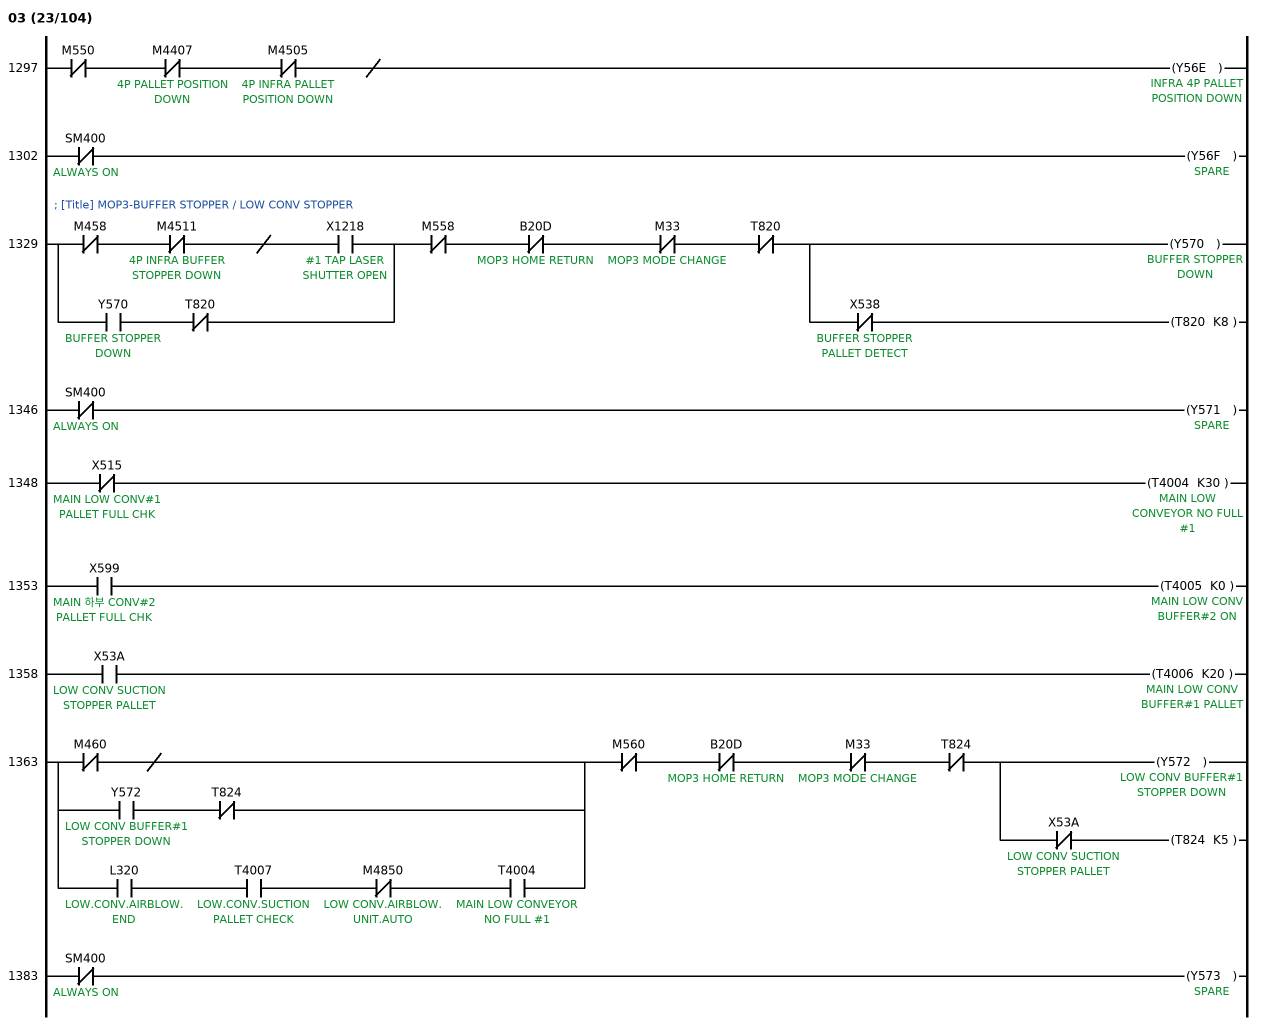
1297  LDI     M550
      ANI     M4407  ; 4P PALLET POSITION DOWN
      ANI     M4505  ; 4P INFRA PALLET POSITION DOWN
      INV
      OUT     Y56E  ; INFRA 4P PALLET POSITION DOWN
1302  LDI     SM400  ; ALWAYS ON
      OUT     Y56F  ; SPARE
; [Title] MOP3-BUFFER STOPPER / LOW CONV STOPPER
1329  LDI     M458
      ANI     M4511  ; 4P INFRA BUFFER STOPPER DOWN
      INV
      AND     X1218  ; #1 TAP LASER SHUTTER OPEN
      LD      Y570  ; BUFFER STOPPER DOWN
      ANI     T820
      ORB
      ANI     M558
      ANI     B20D  ; MOP3 HOME RETURN
      ANI     M33  ; MOP3 MODE CHANGE
      ANI     T820
      OUT     Y570  ; BUFFER STOPPER DOWN
      ANI     X538  ; BUFFER STOPPER PALLET DETECT
      OUT     T820 K8
1346  LDI     SM400  ; ALWAYS ON
      OUT     Y571  ; SPARE
1348  LDI     X515  ; MAIN LOW CONV#1 PALLET FULL CHK
      OUT     T4004 K30  ; MAIN LOW CONVEYOR NO FULL #1
1353  LD      X599  ; MAIN 하부 CONV#2 PALLET FULL CHK
      OUT     T4005 K0  ; MAIN LOW CONV BUFFER#2 ON
1358  LD      X53A  ; LOW CONV SUCTION STOPPER PALLET
      OUT     T4006 K20  ; MAIN LOW CONV BUFFER#1 PALLET
1363  LDI     M460
      INV
      LD      Y572  ; LOW CONV BUFFER#1 STOPPER DOWN
      ANI     T824
      ORB
      LD      L320  ; LOW.CONV.AIRBLOW.END
      AND     T4007  ; LOW.CONV.SUCTION PALLET CHECK
      ANI     M4850  ; LOW CONV.AIRBLOW.UNIT.AUTO
      AND     T4004  ; MAIN LOW CONVEYOR NO FULL #1
      ORB
      ANI     M560
      ANI     B20D  ; MOP3 HOME RETURN
      ANI     M33  ; MOP3 MODE CHANGE
      ANI     T824
      OUT     Y572  ; LOW CONV BUFFER#1 STOPPER DOWN
      ANI     X53A  ; LOW CONV SUCTION STOPPER PALLET
      OUT     T824 K5
1383  LDI     SM400  ; ALWAYS ON
      OUT     Y573  ; SPARE
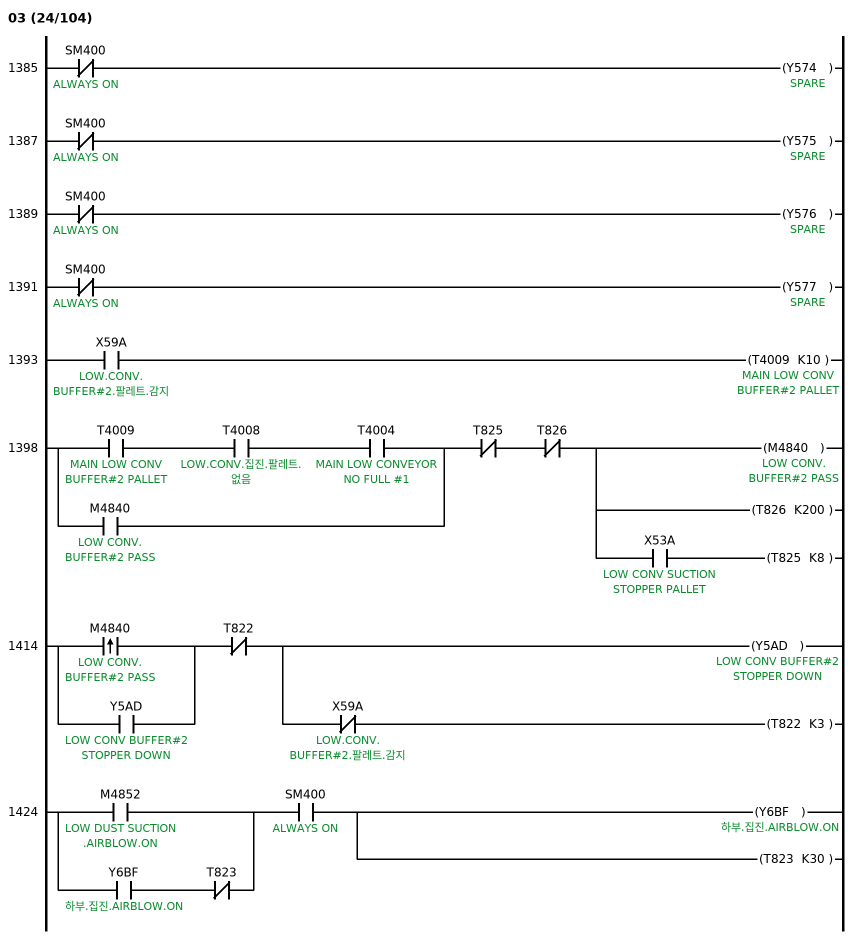
1385  LDI     SM400  ; ALWAYS ON
      OUT     Y574  ; SPARE
1387  LDI     SM400  ; ALWAYS ON
      OUT     Y575  ; SPARE
1389  LDI     SM400  ; ALWAYS ON
      OUT     Y576  ; SPARE
1391  LDI     SM400  ; ALWAYS ON
      OUT     Y577  ; SPARE
1393  LD      X59A  ; LOW.CONV.BUFFER#2.팔레트.감지
      OUT     T4009 K10  ; MAIN LOW CONV BUFFER#2 PALLET
1398  LD      T4009  ; MAIN LOW CONV BUFFER#2 PALLET
      AND     T4008  ; LOW.CONV.집진.팔레트.없음
      AND     T4004  ; MAIN LOW CONVEYOR NO FULL #1
      OR      M4840  ; LOW CONV. BUFFER#2 PASS
      ANI     T825
      ANI     T826
      OUT     M4840  ; LOW CONV. BUFFER#2 PASS
      OUT     T826 K200
      AND     X53A  ; LOW CONV SUCTION STOPPER PALLET
      OUT     T825 K8
1414  LDP     M4840  ; LOW CONV. BUFFER#2 PASS
      OR      Y5AD  ; LOW CONV BUFFER#2 STOPPER DOWN
      ANI     T822
      OUT     Y5AD  ; LOW CONV BUFFER#2 STOPPER DOWN
      ANI     X59A  ; LOW.CONV.BUFFER#2.팔레트.감지
      OUT     T822 K3
1424  LD      M4852  ; LOW DUST SUCTION .AIRBLOW.ON
      LD      Y6BF  ; 하부.집진.AIRBLOW.ON
      ANI     T823
      ORB
      AND     SM400  ; ALWAYS ON
      OUT     Y6BF  ; 하부.집진.AIRBLOW.ON
      OUT     T823 K30
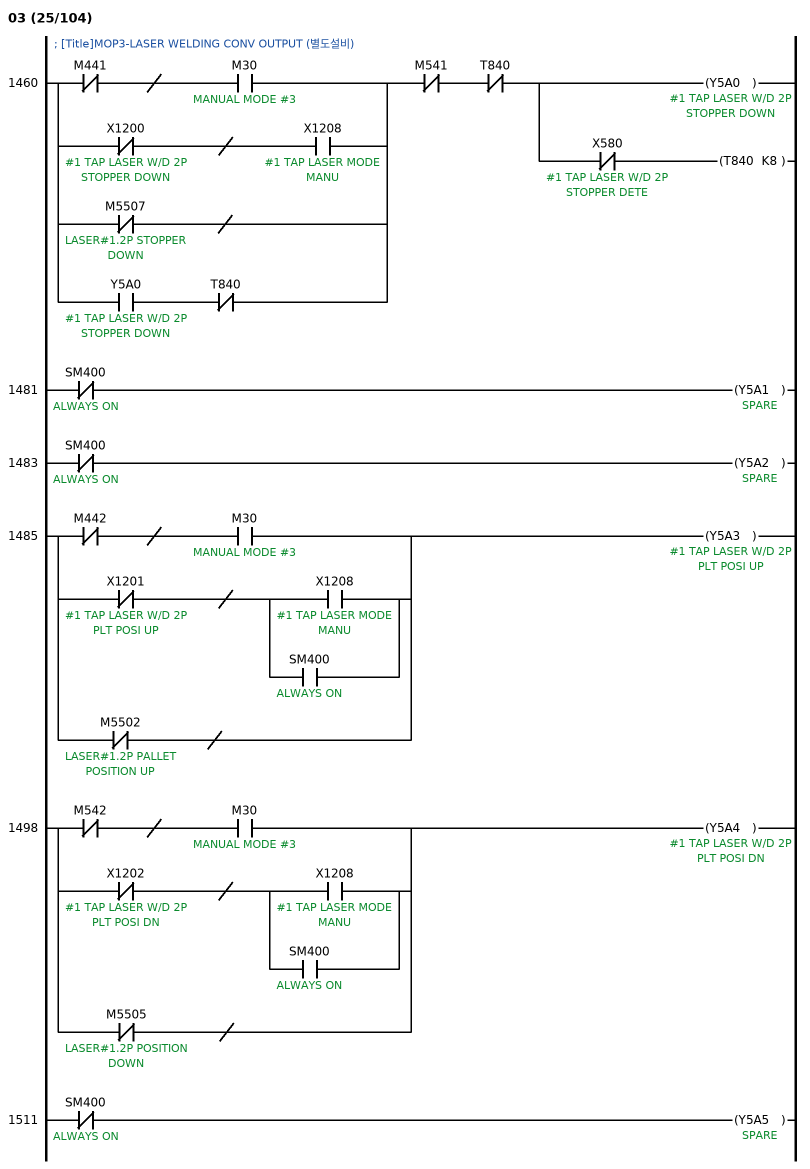
; [Title]MOP3-LASER WELDING CONV OUTPUT (별도설비)
1460  LDI     M441
      INV
      AND     M30  ; MANUAL MODE #3
      LDI     X1200  ; #1 TAP LASER W/D 2P STOPPER DOWN
      INV
      AND     X1208  ; #1 TAP LASER MODE MANU
      ORB
      LDI     M5507  ; LASER#1.2P STOPPER DOWN
      INV
      ORB
      LD      Y5A0  ; #1 TAP LASER W/D 2P STOPPER DOWN
      ANI     T840
      ORB
      ANI     M541
      ANI     T840
      OUT     Y5A0  ; #1 TAP LASER W/D 2P STOPPER DOWN
      ANI     X580  ; #1 TAP LASER W/D 2P STOPPER DETE
      OUT     T840 K8
1481  LDI     SM400  ; ALWAYS ON
      OUT     Y5A1  ; SPARE
1483  LDI     SM400  ; ALWAYS ON
      OUT     Y5A2  ; SPARE
1485  LDI     M442
      INV
      AND     M30  ; MANUAL MODE #3
      LDI     X1201  ; #1 TAP LASER W/D 2P PLT POSI UP
      INV
      LD      X1208  ; #1 TAP LASER MODE MANU
      OR      SM400  ; ALWAYS ON
      ANB
      ORB
      LDI     M5502  ; LASER#1.2P PALLET POSITION UP
      INV
      ORB
      OUT     Y5A3  ; #1 TAP LASER W/D 2P PLT POSI UP
1498  LDI     M542
      INV
      AND     M30  ; MANUAL MODE #3
      LDI     X1202  ; #1 TAP LASER W/D 2P PLT POSI DN
      INV
      LD      X1208  ; #1 TAP LASER MODE MANU
      OR      SM400  ; ALWAYS ON
      ANB
      ORB
      LDI     M5505  ; LASER#1.2P POSITION DOWN
      INV
      ORB
      OUT     Y5A4  ; #1 TAP LASER W/D 2P PLT POSI DN
1511  LDI     SM400  ; ALWAYS ON
      OUT     Y5A5  ; SPARE
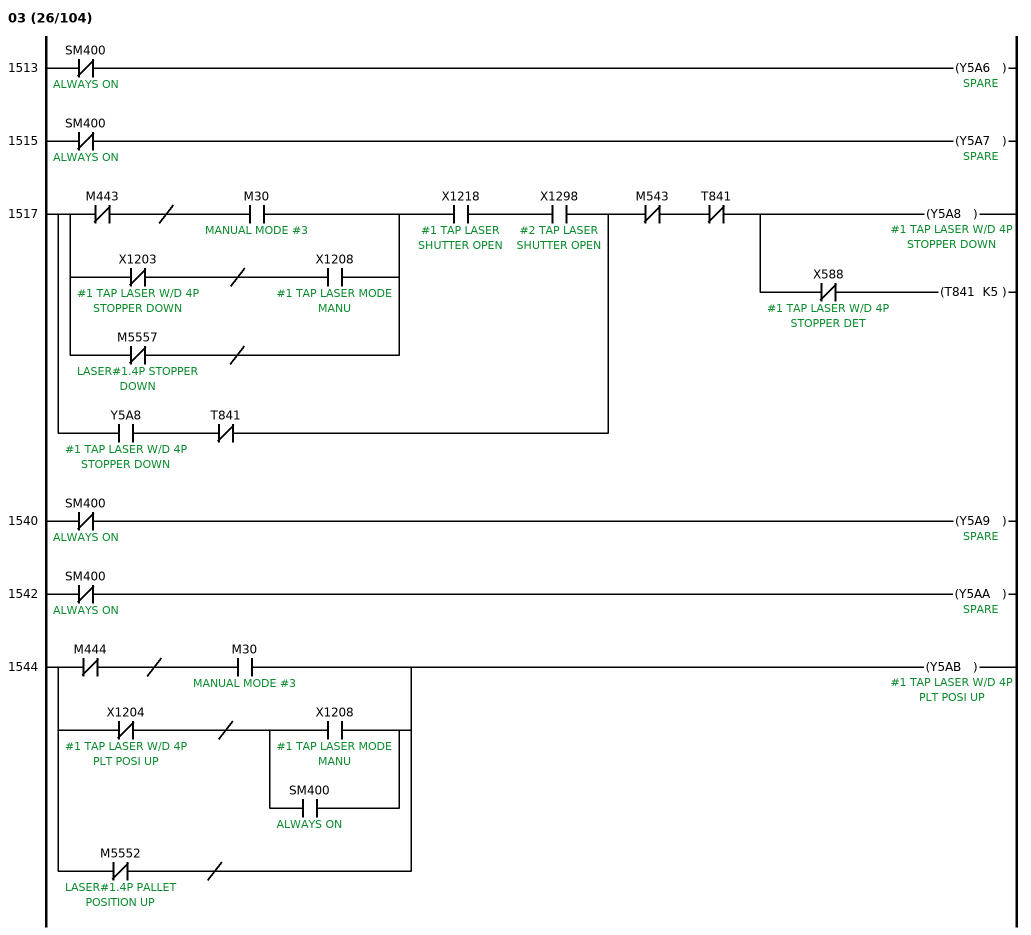
1513  LDI     SM400  ; ALWAYS ON
      OUT     Y5A6  ; SPARE
1515  LDI     SM400  ; ALWAYS ON
      OUT     Y5A7  ; SPARE
1517  LDI     M443
      INV
      AND     M30  ; MANUAL MODE #3
      LDI     X1203  ; #1 TAP LASER W/D 4P STOPPER DOWN
      INV
      AND     X1208  ; #1 TAP LASER MODE MANU
      ORB
      LDI     M5557  ; LASER#1.4P STOPPER DOWN
      INV
      ORB
      AND     X1218  ; #1 TAP LASER SHUTTER OPEN
      AND     X1298  ; #2 TAP LASER SHUTTER OPEN
      LD      Y5A8  ; #1 TAP LASER W/D 4P STOPPER DOWN
      ANI     T841
      ORB
      ANI     M543
      ANI     T841
      OUT     Y5A8  ; #1 TAP LASER W/D 4P STOPPER DOWN
      ANI     X588  ; #1 TAP LASER W/D 4P STOPPER DET
      OUT     T841 K5
1540  LDI     SM400  ; ALWAYS ON
      OUT     Y5A9  ; SPARE
1542  LDI     SM400  ; ALWAYS ON
      OUT     Y5AA  ; SPARE
1544  LDI     M444
      INV
      AND     M30  ; MANUAL MODE #3
      LDI     X1204  ; #1 TAP LASER W/D 4P PLT POSI UP
      INV
      LD      X1208  ; #1 TAP LASER MODE MANU
      OR      SM400  ; ALWAYS ON
      ANB
      ORB
      LDI     M5552  ; LASER#1.4P PALLET POSITION UP
      INV
      ORB
      OUT     Y5AB  ; #1 TAP LASER W/D 4P PLT POSI UP
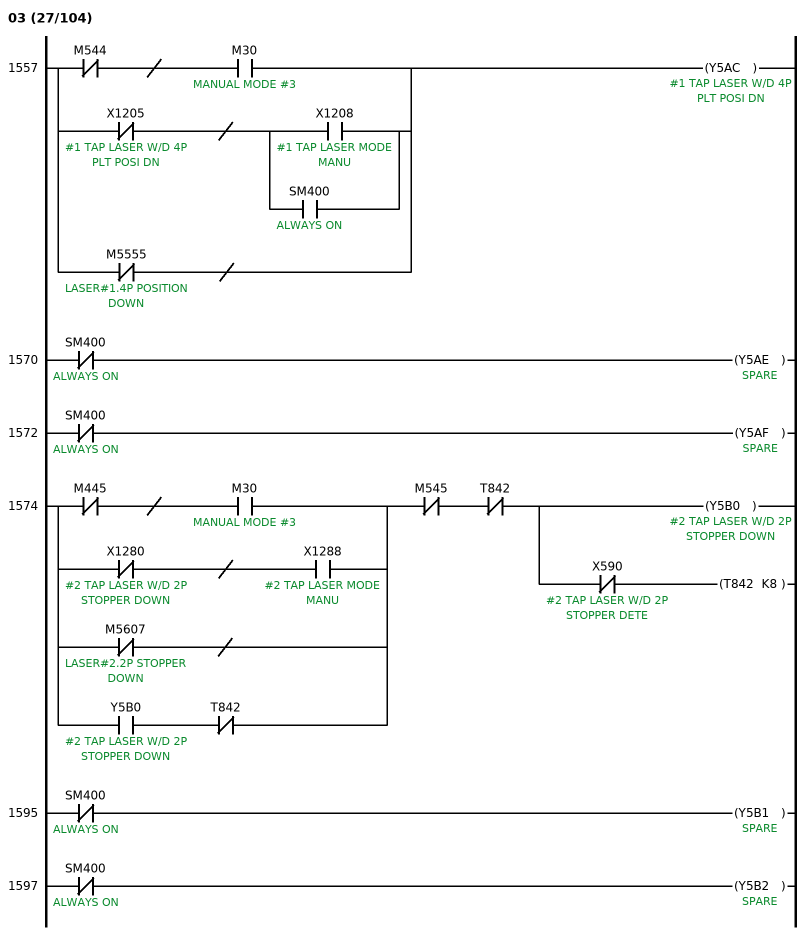
1557  LDI     M544
      INV
      AND     M30  ; MANUAL MODE #3
      LDI     X1205  ; #1 TAP LASER W/D 4P PLT POSI DN
      INV
      LD      X1208  ; #1 TAP LASER MODE MANU
      OR      SM400  ; ALWAYS ON
      ANB
      ORB
      LDI     M5555  ; LASER#1.4P POSITION DOWN
      INV
      ORB
      OUT     Y5AC  ; #1 TAP LASER W/D 4P PLT POSI DN
1570  LDI     SM400  ; ALWAYS ON
      OUT     Y5AE  ; SPARE
1572  LDI     SM400  ; ALWAYS ON
      OUT     Y5AF  ; SPARE
1574  LDI     M445
      INV
      AND     M30  ; MANUAL MODE #3
      LDI     X1280  ; #2 TAP LASER W/D 2P STOPPER DOWN
      INV
      AND     X1288  ; #2 TAP LASER MODE MANU
      ORB
      LDI     M5607  ; LASER#2.2P STOPPER DOWN
      INV
      ORB
      LD      Y5B0  ; #2 TAP LASER W/D 2P STOPPER DOWN
      ANI     T842
      ORB
      ANI     M545
      ANI     T842
      OUT     Y5B0  ; #2 TAP LASER W/D 2P STOPPER DOWN
      ANI     X590  ; #2 TAP LASER W/D 2P STOPPER DETE
      OUT     T842 K8
1595  LDI     SM400  ; ALWAYS ON
      OUT     Y5B1  ; SPARE
1597  LDI     SM400  ; ALWAYS ON
      OUT     Y5B2  ; SPARE
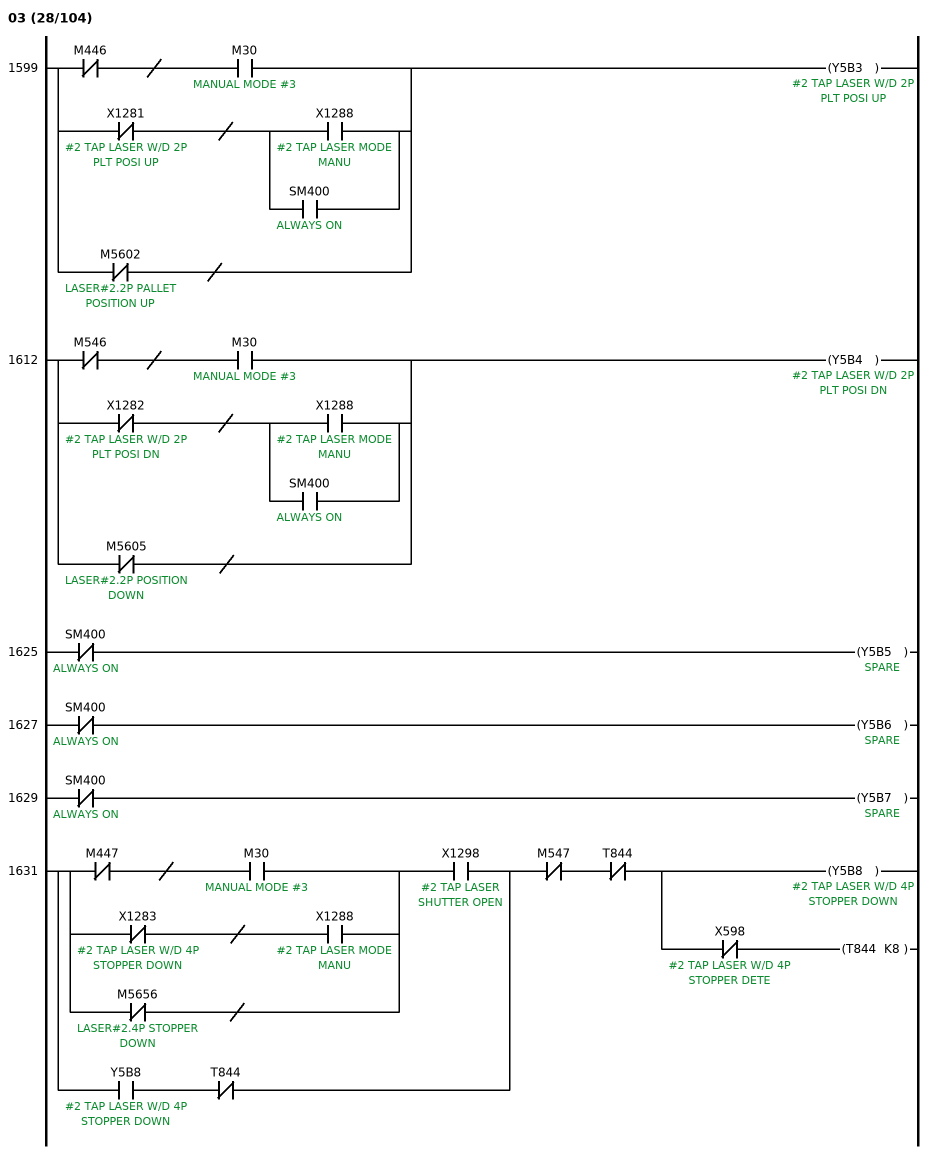
1599  LDI     M446
      INV
      AND     M30  ; MANUAL MODE #3
      LDI     X1281  ; #2 TAP LASER W/D 2P PLT POSI UP
      INV
      LD      X1288  ; #2 TAP LASER MODE MANU
      OR      SM400  ; ALWAYS ON
      ANB
      ORB
      LDI     M5602  ; LASER#2.2P PALLET POSITION UP
      INV
      ORB
      OUT     Y5B3  ; #2 TAP LASER W/D 2P PLT POSI UP
1612  LDI     M546
      INV
      AND     M30  ; MANUAL MODE #3
      LDI     X1282  ; #2 TAP LASER W/D 2P PLT POSI DN
      INV
      LD      X1288  ; #2 TAP LASER MODE MANU
      OR      SM400  ; ALWAYS ON
      ANB
      ORB
      LDI     M5605  ; LASER#2.2P POSITION DOWN
      INV
      ORB
      OUT     Y5B4  ; #2 TAP LASER W/D 2P PLT POSI DN
1625  LDI     SM400  ; ALWAYS ON
      OUT     Y5B5  ; SPARE
1627  LDI     SM400  ; ALWAYS ON
      OUT     Y5B6  ; SPARE
1629  LDI     SM400  ; ALWAYS ON
      OUT     Y5B7  ; SPARE
1631  LDI     M447
      INV
      AND     M30  ; MANUAL MODE #3
      LDI     X1283  ; #2 TAP LASER W/D 4P STOPPER DOWN
      INV
      AND     X1288  ; #2 TAP LASER MODE MANU
      ORB
      LDI     M5656  ; LASER#2.4P STOPPER DOWN
      INV
      ORB
      AND     X1298  ; #2 TAP LASER SHUTTER OPEN
      LD      Y5B8  ; #2 TAP LASER W/D 4P STOPPER DOWN
      ANI     T844
      ORB
      ANI     M547
      ANI     T844
      OUT     Y5B8  ; #2 TAP LASER W/D 4P STOPPER DOWN
      ANI     X598  ; #2 TAP LASER W/D 4P STOPPER DETE
      OUT     T844 K8
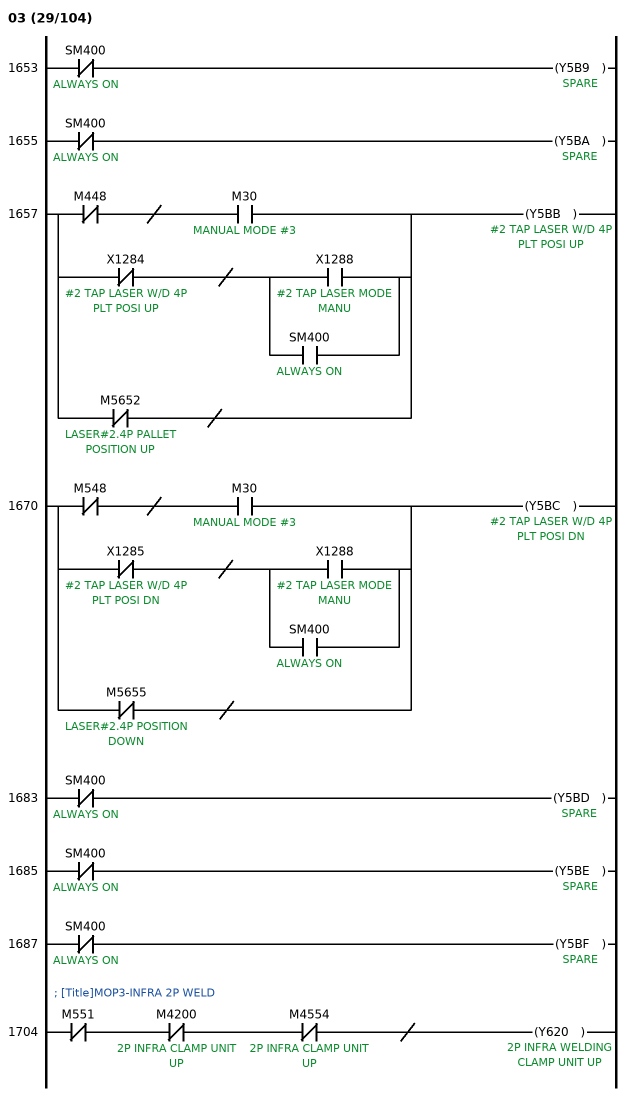
1653  LDI     SM400  ; ALWAYS ON
      OUT     Y5B9  ; SPARE
1655  LDI     SM400  ; ALWAYS ON
      OUT     Y5BA  ; SPARE
1657  LDI     M448
      INV
      AND     M30  ; MANUAL MODE #3
      LDI     X1284  ; #2 TAP LASER W/D 4P PLT POSI UP
      INV
      LD      X1288  ; #2 TAP LASER MODE MANU
      OR      SM400  ; ALWAYS ON
      ANB
      ORB
      LDI     M5652  ; LASER#2.4P PALLET POSITION UP
      INV
      ORB
      OUT     Y5BB  ; #2 TAP LASER W/D 4P PLT POSI UP
1670  LDI     M548
      INV
      AND     M30  ; MANUAL MODE #3
      LDI     X1285  ; #2 TAP LASER W/D 4P PLT POSI DN
      INV
      LD      X1288  ; #2 TAP LASER MODE MANU
      OR      SM400  ; ALWAYS ON
      ANB
      ORB
      LDI     M5655  ; LASER#2.4P POSITION DOWN
      INV
      ORB
      OUT     Y5BC  ; #2 TAP LASER W/D 4P PLT POSI DN
1683  LDI     SM400  ; ALWAYS ON
      OUT     Y5BD  ; SPARE
1685  LDI     SM400  ; ALWAYS ON
      OUT     Y5BE  ; SPARE
1687  LDI     SM400  ; ALWAYS ON
      OUT     Y5BF  ; SPARE
; [Title]MOP3-INFRA 2P WELD
1704  LDI     M551
      ANI     M4200  ; 2P INFRA CLAMP UNIT UP
      ANI     M4554  ; 2P INFRA CLAMP UNIT UP
      INV
      OUT     Y620  ; 2P INFRA WELDING CLAMP UNIT UP
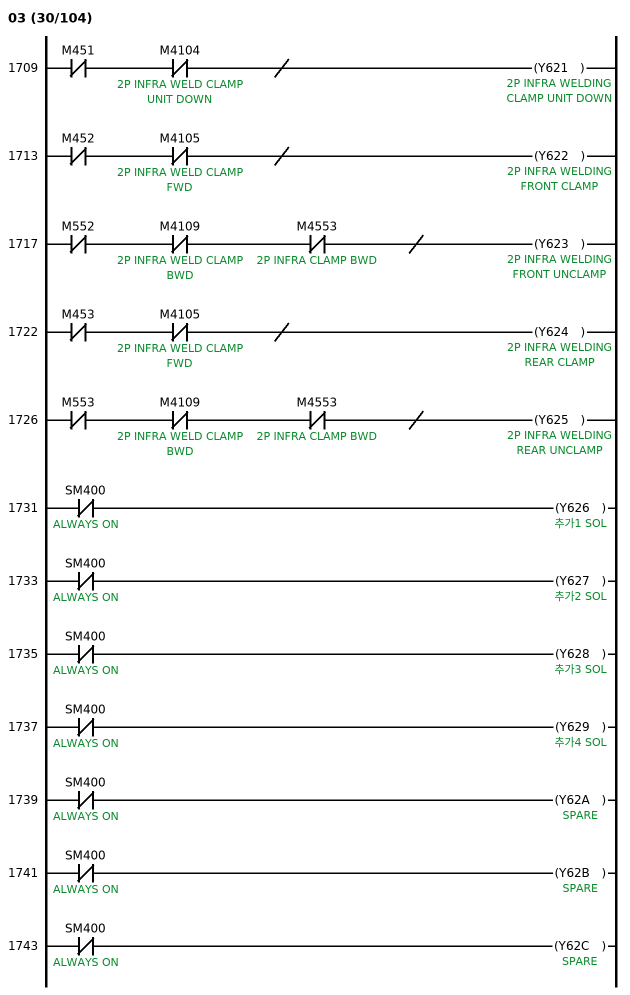
1709  LDI     M451
      ANI     M4104  ; 2P INFRA WELD CLAMP UNIT DOWN
      INV
      OUT     Y621  ; 2P INFRA WELDING CLAMP UNIT DOWN
1713  LDI     M452
      ANI     M4105  ; 2P INFRA WELD CLAMP FWD
      INV
      OUT     Y622  ; 2P INFRA WELDING FRONT CLAMP
1717  LDI     M552
      ANI     M4109  ; 2P INFRA WELD CLAMP BWD
      ANI     M4553  ; 2P INFRA CLAMP BWD
      INV
      OUT     Y623  ; 2P INFRA WELDING FRONT UNCLAMP
1722  LDI     M453
      ANI     M4105  ; 2P INFRA WELD CLAMP FWD
      INV
      OUT     Y624  ; 2P INFRA WELDING REAR CLAMP
1726  LDI     M553
      ANI     M4109  ; 2P INFRA WELD CLAMP BWD
      ANI     M4553  ; 2P INFRA CLAMP BWD
      INV
      OUT     Y625  ; 2P INFRA WELDING REAR UNCLAMP
1731  LDI     SM400  ; ALWAYS ON
      OUT     Y626  ; 추가1 SOL
1733  LDI     SM400  ; ALWAYS ON
      OUT     Y627  ; 추가2 SOL
1735  LDI     SM400  ; ALWAYS ON
      OUT     Y628  ; 추가3 SOL
1737  LDI     SM400  ; ALWAYS ON
      OUT     Y629  ; 추가4 SOL
1739  LDI     SM400  ; ALWAYS ON
      OUT     Y62A  ; SPARE
1741  LDI     SM400  ; ALWAYS ON
      OUT     Y62B  ; SPARE
1743  LDI     SM400  ; ALWAYS ON
      OUT     Y62C  ; SPARE
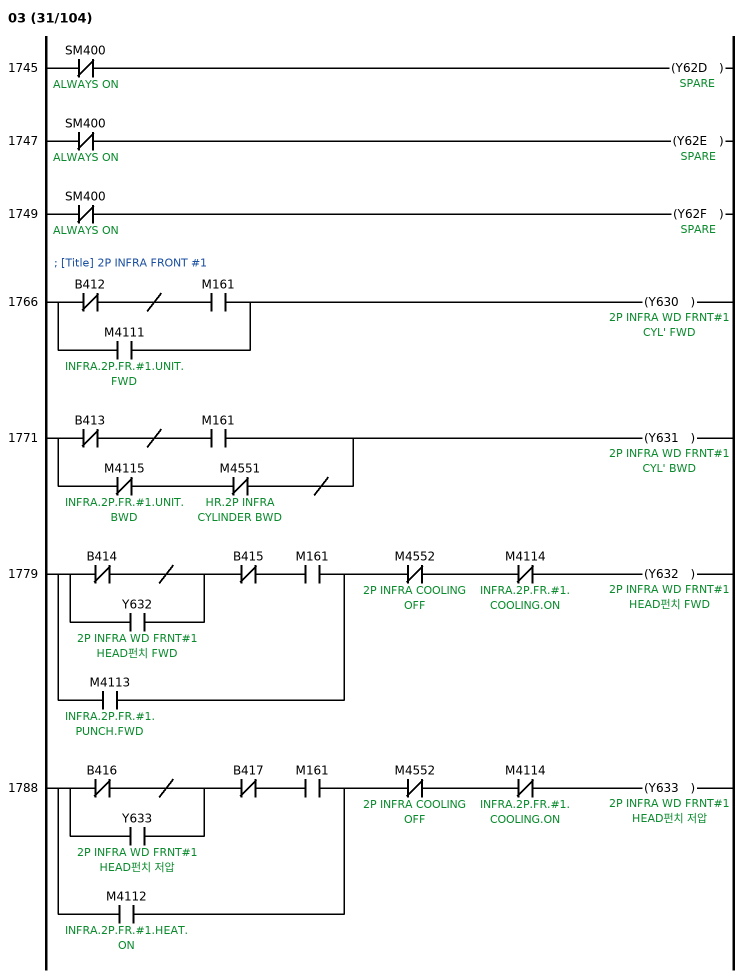
1745  LDI     SM400  ; ALWAYS ON
      OUT     Y62D  ; SPARE
1747  LDI     SM400  ; ALWAYS ON
      OUT     Y62E  ; SPARE
1749  LDI     SM400  ; ALWAYS ON
      OUT     Y62F  ; SPARE
; [Title] 2P INFRA FRONT #1
1766  LDI     B412
      INV
      AND     M161
      OR      M4111  ; INFRA.2P.FR.#1.UNIT.FWD
      OUT     Y630  ; 2P INFRA WD FRNT#1 CYL' FWD
1771  LDI     B413
      INV
      AND     M161
      LDI     M4115  ; INFRA.2P.FR.#1.UNIT.BWD
      ANI     M4551  ; HR.2P INFRA CYLINDER BWD
      INV
      ORB
      OUT     Y631  ; 2P INFRA WD FRNT#1 CYL' BWD
1779  LDI     B414
      INV
      OR      Y632  ; 2P INFRA WD FRNT#1 HEAD펀치 FWD
      ANI     B415
      AND     M161
      OR      M4113  ; INFRA.2P.FR.#1.PUNCH.FWD
      ANI     M4552  ; 2P INFRA COOLING OFF
      ANI     M4114  ; INFRA.2P.FR.#1.COOLING.ON
      OUT     Y632  ; 2P INFRA WD FRNT#1 HEAD펀치 FWD
1788  LDI     B416
      INV
      OR      Y633  ; 2P INFRA WD FRNT#1 HEAD펀치 저압
      ANI     B417
      AND     M161
      OR      M4112  ; INFRA.2P.FR.#1.HEAT.ON
      ANI     M4552  ; 2P INFRA COOLING OFF
      ANI     M4114  ; INFRA.2P.FR.#1.COOLING.ON
      OUT     Y633  ; 2P INFRA WD FRNT#1 HEAD펀치 저압
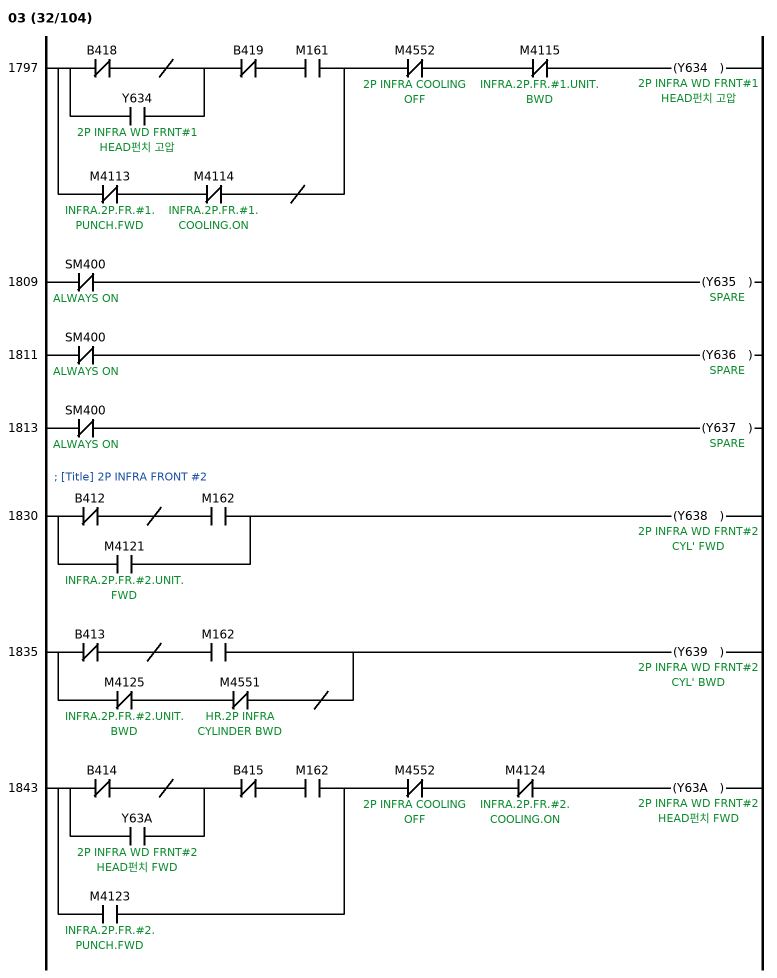
1797  LDI     B418
      INV
      OR      Y634  ; 2P INFRA WD FRNT#1 HEAD펀치 고압
      ANI     B419
      AND     M161
      LDI     M4113  ; INFRA.2P.FR.#1.PUNCH.FWD
      ANI     M4114  ; INFRA.2P.FR.#1.COOLING.ON
      INV
      ORB
      ANI     M4552  ; 2P INFRA COOLING OFF
      ANI     M4115  ; INFRA.2P.FR.#1.UNIT.BWD
      OUT     Y634  ; 2P INFRA WD FRNT#1 HEAD펀치 고압
1809  LDI     SM400  ; ALWAYS ON
      OUT     Y635  ; SPARE
1811  LDI     SM400  ; ALWAYS ON
      OUT     Y636  ; SPARE
1813  LDI     SM400  ; ALWAYS ON
      OUT     Y637  ; SPARE
; [Title] 2P INFRA FRONT #2
1830  LDI     B412
      INV
      AND     M162
      OR      M4121  ; INFRA.2P.FR.#2.UNIT.FWD
      OUT     Y638  ; 2P INFRA WD FRNT#2 CYL' FWD
1835  LDI     B413
      INV
      AND     M162
      LDI     M4125  ; INFRA.2P.FR.#2.UNIT.BWD
      ANI     M4551  ; HR.2P INFRA CYLINDER BWD
      INV
      ORB
      OUT     Y639  ; 2P INFRA WD FRNT#2 CYL' BWD
1843  LDI     B414
      INV
      OR      Y63A  ; 2P INFRA WD FRNT#2 HEAD펀치 FWD
      ANI     B415
      AND     M162
      OR      M4123  ; INFRA.2P.FR.#2.PUNCH.FWD
      ANI     M4552  ; 2P INFRA COOLING OFF
      ANI     M4124  ; INFRA.2P.FR.#2.COOLING.ON
      OUT     Y63A  ; 2P INFRA WD FRNT#2 HEAD펀치 FWD
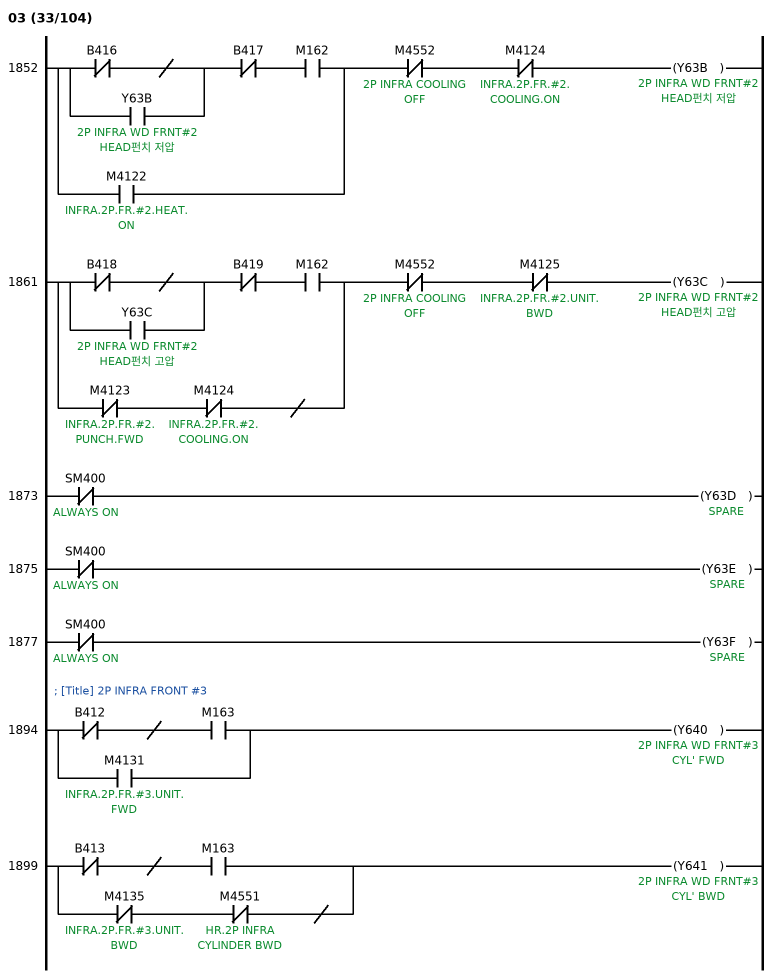
1852  LDI     B416
      INV
      OR      Y63B  ; 2P INFRA WD FRNT#2 HEAD펀치 저압
      ANI     B417
      AND     M162
      OR      M4122  ; INFRA.2P.FR.#2.HEAT.ON
      ANI     M4552  ; 2P INFRA COOLING OFF
      ANI     M4124  ; INFRA.2P.FR.#2.COOLING.ON
      OUT     Y63B  ; 2P INFRA WD FRNT#2 HEAD펀치 저압
1861  LDI     B418
      INV
      OR      Y63C  ; 2P INFRA WD FRNT#2 HEAD펀치 고압
      ANI     B419
      AND     M162
      LDI     M4123  ; INFRA.2P.FR.#2.PUNCH.FWD
      ANI     M4124  ; INFRA.2P.FR.#2.COOLING.ON
      INV
      ORB
      ANI     M4552  ; 2P INFRA COOLING OFF
      ANI     M4125  ; INFRA.2P.FR.#2.UNIT.BWD
      OUT     Y63C  ; 2P INFRA WD FRNT#2 HEAD펀치 고압
1873  LDI     SM400  ; ALWAYS ON
      OUT     Y63D  ; SPARE
1875  LDI     SM400  ; ALWAYS ON
      OUT     Y63E  ; SPARE
1877  LDI     SM400  ; ALWAYS ON
      OUT     Y63F  ; SPARE
; [Title] 2P INFRA FRONT #3
1894  LDI     B412
      INV
      AND     M163
      OR      M4131  ; INFRA.2P.FR.#3.UNIT.FWD
      OUT     Y640  ; 2P INFRA WD FRNT#3 CYL' FWD
1899  LDI     B413
      INV
      AND     M163
      LDI     M4135  ; INFRA.2P.FR.#3.UNIT.BWD
      ANI     M4551  ; HR.2P INFRA CYLINDER BWD
      INV
      ORB
      OUT     Y641  ; 2P INFRA WD FRNT#3 CYL' BWD
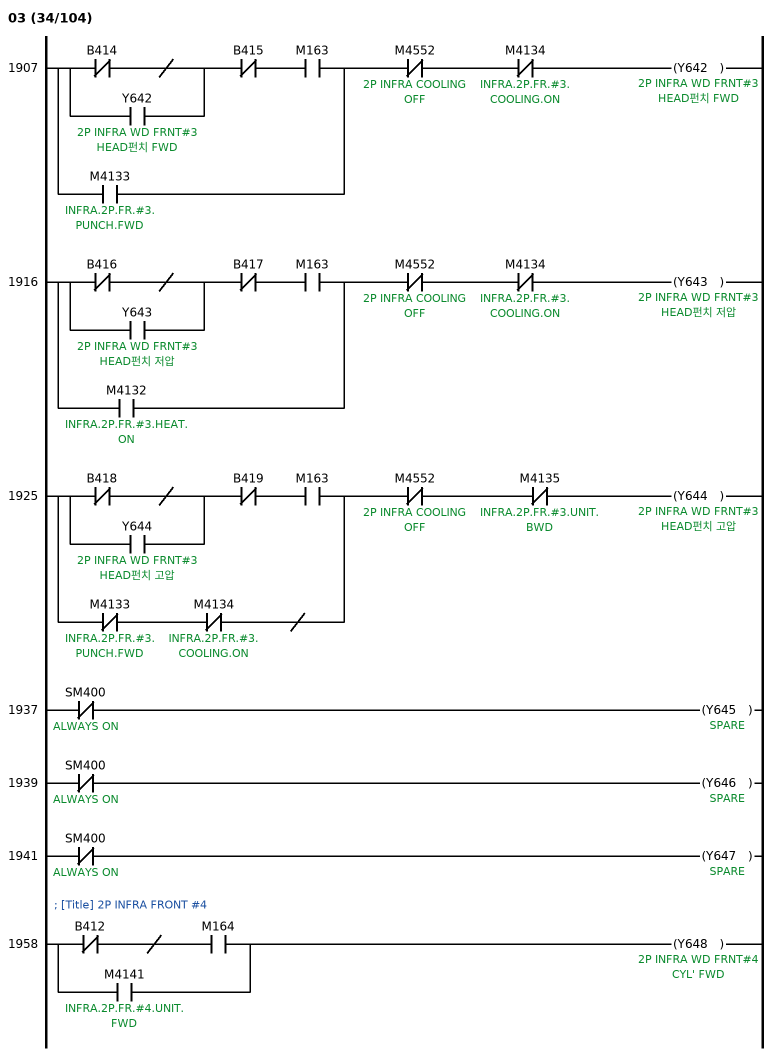
1907  LDI     B414
      INV
      OR      Y642  ; 2P INFRA WD FRNT#3 HEAD펀치 FWD
      ANI     B415
      AND     M163
      OR      M4133  ; INFRA.2P.FR.#3.PUNCH.FWD
      ANI     M4552  ; 2P INFRA COOLING OFF
      ANI     M4134  ; INFRA.2P.FR.#3.COOLING.ON
      OUT     Y642  ; 2P INFRA WD FRNT#3 HEAD펀치 FWD
1916  LDI     B416
      INV
      OR      Y643  ; 2P INFRA WD FRNT#3 HEAD펀치 저압
      ANI     B417
      AND     M163
      OR      M4132  ; INFRA.2P.FR.#3.HEAT.ON
      ANI     M4552  ; 2P INFRA COOLING OFF
      ANI     M4134  ; INFRA.2P.FR.#3.COOLING.ON
      OUT     Y643  ; 2P INFRA WD FRNT#3 HEAD펀치 저압
1925  LDI     B418
      INV
      OR      Y644  ; 2P INFRA WD FRNT#3 HEAD펀치 고압
      ANI     B419
      AND     M163
      LDI     M4133  ; INFRA.2P.FR.#3.PUNCH.FWD
      ANI     M4134  ; INFRA.2P.FR.#3.COOLING.ON
      INV
      ORB
      ANI     M4552  ; 2P INFRA COOLING OFF
      ANI     M4135  ; INFRA.2P.FR.#3.UNIT.BWD
      OUT     Y644  ; 2P INFRA WD FRNT#3 HEAD펀치 고압
1937  LDI     SM400  ; ALWAYS ON
      OUT     Y645  ; SPARE
1939  LDI     SM400  ; ALWAYS ON
      OUT     Y646  ; SPARE
1941  LDI     SM400  ; ALWAYS ON
      OUT     Y647  ; SPARE
; [Title] 2P INFRA FRONT #4
1958  LDI     B412
      INV
      AND     M164
      OR      M4141  ; INFRA.2P.FR.#4.UNIT.FWD
      OUT     Y648  ; 2P INFRA WD FRNT#4 CYL' FWD
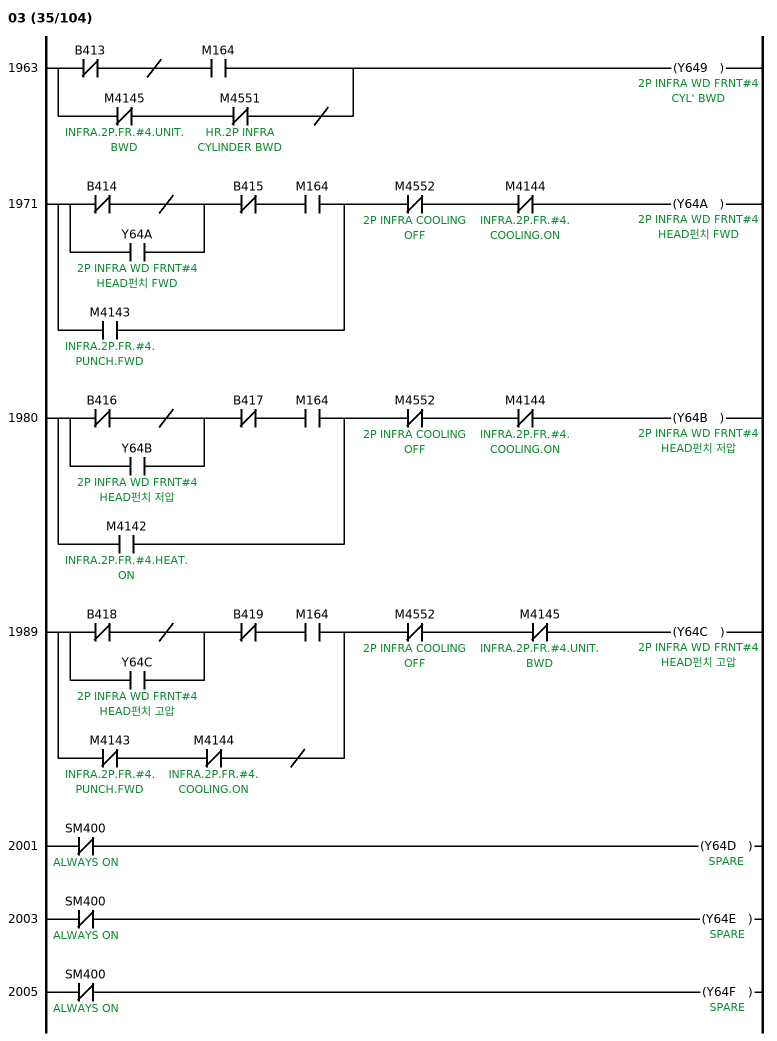
1963  LDI     B413
      INV
      AND     M164
      LDI     M4145  ; INFRA.2P.FR.#4.UNIT.BWD
      ANI     M4551  ; HR.2P INFRA CYLINDER BWD
      INV
      ORB
      OUT     Y649  ; 2P INFRA WD FRNT#4 CYL' BWD
1971  LDI     B414
      INV
      OR      Y64A  ; 2P INFRA WD FRNT#4 HEAD펀치 FWD
      ANI     B415
      AND     M164
      OR      M4143  ; INFRA.2P.FR.#4.PUNCH.FWD
      ANI     M4552  ; 2P INFRA COOLING OFF
      ANI     M4144  ; INFRA.2P.FR.#4.COOLING.ON
      OUT     Y64A  ; 2P INFRA WD FRNT#4 HEAD펀치 FWD
1980  LDI     B416
      INV
      OR      Y64B  ; 2P INFRA WD FRNT#4 HEAD펀치 저압
      ANI     B417
      AND     M164
      OR      M4142  ; INFRA.2P.FR.#4.HEAT.ON
      ANI     M4552  ; 2P INFRA COOLING OFF
      ANI     M4144  ; INFRA.2P.FR.#4.COOLING.ON
      OUT     Y64B  ; 2P INFRA WD FRNT#4 HEAD펀치 저압
1989  LDI     B418
      INV
      OR      Y64C  ; 2P INFRA WD FRNT#4 HEAD펀치 고압
      ANI     B419
      AND     M164
      LDI     M4143  ; INFRA.2P.FR.#4.PUNCH.FWD
      ANI     M4144  ; INFRA.2P.FR.#4.COOLING.ON
      INV
      ORB
      ANI     M4552  ; 2P INFRA COOLING OFF
      ANI     M4145  ; INFRA.2P.FR.#4.UNIT.BWD
      OUT     Y64C  ; 2P INFRA WD FRNT#4 HEAD펀치 고압
2001  LDI     SM400  ; ALWAYS ON
      OUT     Y64D  ; SPARE
2003  LDI     SM400  ; ALWAYS ON
      OUT     Y64E  ; SPARE
2005  LDI     SM400  ; ALWAYS ON
      OUT     Y64F  ; SPARE
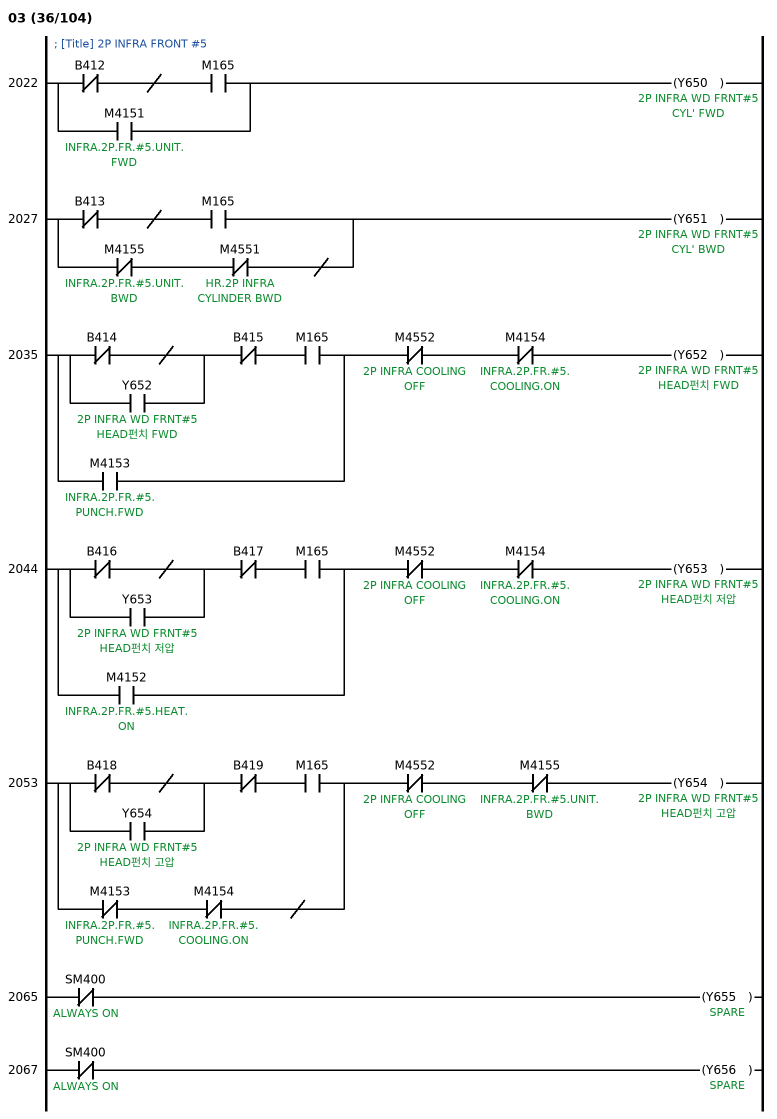
; [Title] 2P INFRA FRONT #5
2022  LDI     B412
      INV
      AND     M165
      OR      M4151  ; INFRA.2P.FR.#5.UNIT.FWD
      OUT     Y650  ; 2P INFRA WD FRNT#5 CYL' FWD
2027  LDI     B413
      INV
      AND     M165
      LDI     M4155  ; INFRA.2P.FR.#5.UNIT.BWD
      ANI     M4551  ; HR.2P INFRA CYLINDER BWD
      INV
      ORB
      OUT     Y651  ; 2P INFRA WD FRNT#5 CYL' BWD
2035  LDI     B414
      INV
      OR      Y652  ; 2P INFRA WD FRNT#5 HEAD펀치 FWD
      ANI     B415
      AND     M165
      OR      M4153  ; INFRA.2P.FR.#5.PUNCH.FWD
      ANI     M4552  ; 2P INFRA COOLING OFF
      ANI     M4154  ; INFRA.2P.FR.#5.COOLING.ON
      OUT     Y652  ; 2P INFRA WD FRNT#5 HEAD펀치 FWD
2044  LDI     B416
      INV
      OR      Y653  ; 2P INFRA WD FRNT#5 HEAD펀치 저압
      ANI     B417
      AND     M165
      OR      M4152  ; INFRA.2P.FR.#5.HEAT.ON
      ANI     M4552  ; 2P INFRA COOLING OFF
      ANI     M4154  ; INFRA.2P.FR.#5.COOLING.ON
      OUT     Y653  ; 2P INFRA WD FRNT#5 HEAD펀치 저압
2053  LDI     B418
      INV
      OR      Y654  ; 2P INFRA WD FRNT#5 HEAD펀치 고압
      ANI     B419
      AND     M165
      LDI     M4153  ; INFRA.2P.FR.#5.PUNCH.FWD
      ANI     M4154  ; INFRA.2P.FR.#5.COOLING.ON
      INV
      ORB
      ANI     M4552  ; 2P INFRA COOLING OFF
      ANI     M4155  ; INFRA.2P.FR.#5.UNIT.BWD
      OUT     Y654  ; 2P INFRA WD FRNT#5 HEAD펀치 고압
2065  LDI     SM400  ; ALWAYS ON
      OUT     Y655  ; SPARE
2067  LDI     SM400  ; ALWAYS ON
      OUT     Y656  ; SPARE
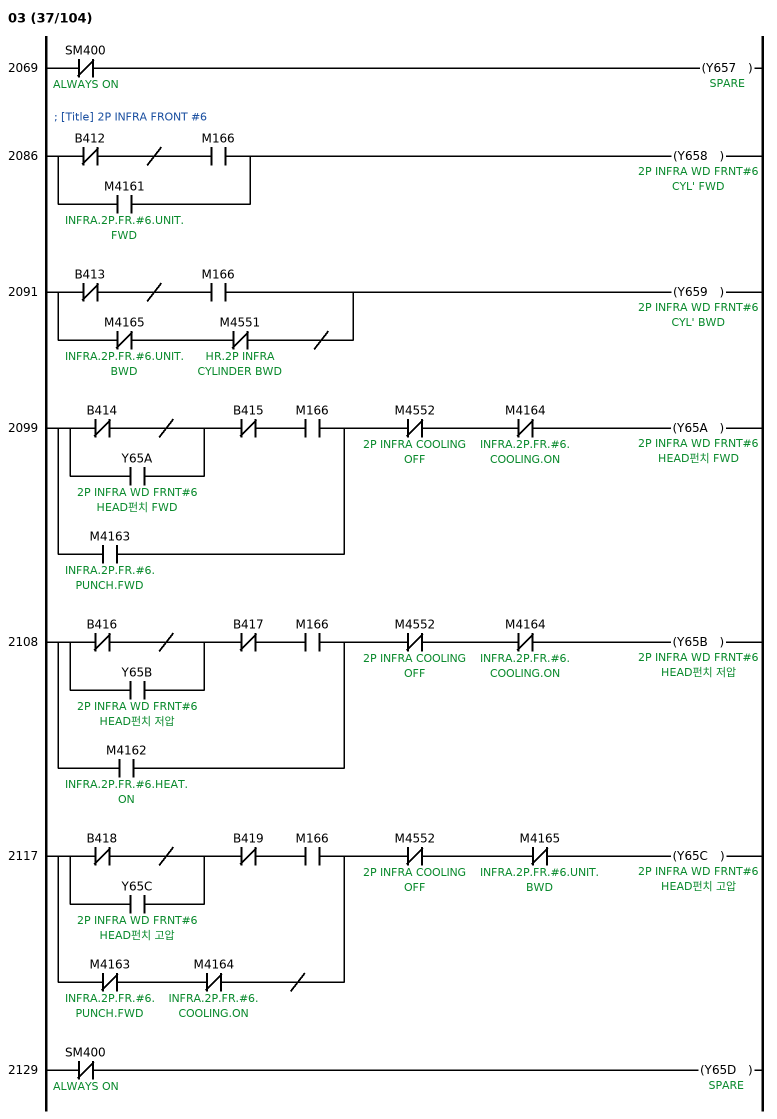
2069  LDI     SM400  ; ALWAYS ON
      OUT     Y657  ; SPARE
; [Title] 2P INFRA FRONT #6
2086  LDI     B412
      INV
      AND     M166
      OR      M4161  ; INFRA.2P.FR.#6.UNIT.FWD
      OUT     Y658  ; 2P INFRA WD FRNT#6 CYL' FWD
2091  LDI     B413
      INV
      AND     M166
      LDI     M4165  ; INFRA.2P.FR.#6.UNIT.BWD
      ANI     M4551  ; HR.2P INFRA CYLINDER BWD
      INV
      ORB
      OUT     Y659  ; 2P INFRA WD FRNT#6 CYL' BWD
2099  LDI     B414
      INV
      OR      Y65A  ; 2P INFRA WD FRNT#6 HEAD펀치 FWD
      ANI     B415
      AND     M166
      OR      M4163  ; INFRA.2P.FR.#6.PUNCH.FWD
      ANI     M4552  ; 2P INFRA COOLING OFF
      ANI     M4164  ; INFRA.2P.FR.#6.COOLING.ON
      OUT     Y65A  ; 2P INFRA WD FRNT#6 HEAD펀치 FWD
2108  LDI     B416
      INV
      OR      Y65B  ; 2P INFRA WD FRNT#6 HEAD펀치 저압
      ANI     B417
      AND     M166
      OR      M4162  ; INFRA.2P.FR.#6.HEAT.ON
      ANI     M4552  ; 2P INFRA COOLING OFF
      ANI     M4164  ; INFRA.2P.FR.#6.COOLING.ON
      OUT     Y65B  ; 2P INFRA WD FRNT#6 HEAD펀치 저압
2117  LDI     B418
      INV
      OR      Y65C  ; 2P INFRA WD FRNT#6 HEAD펀치 고압
      ANI     B419
      AND     M166
      LDI     M4163  ; INFRA.2P.FR.#6.PUNCH.FWD
      ANI     M4164  ; INFRA.2P.FR.#6.COOLING.ON
      INV
      ORB
      ANI     M4552  ; 2P INFRA COOLING OFF
      ANI     M4165  ; INFRA.2P.FR.#6.UNIT.BWD
      OUT     Y65C  ; 2P INFRA WD FRNT#6 HEAD펀치 고압
2129  LDI     SM400  ; ALWAYS ON
      OUT     Y65D  ; SPARE
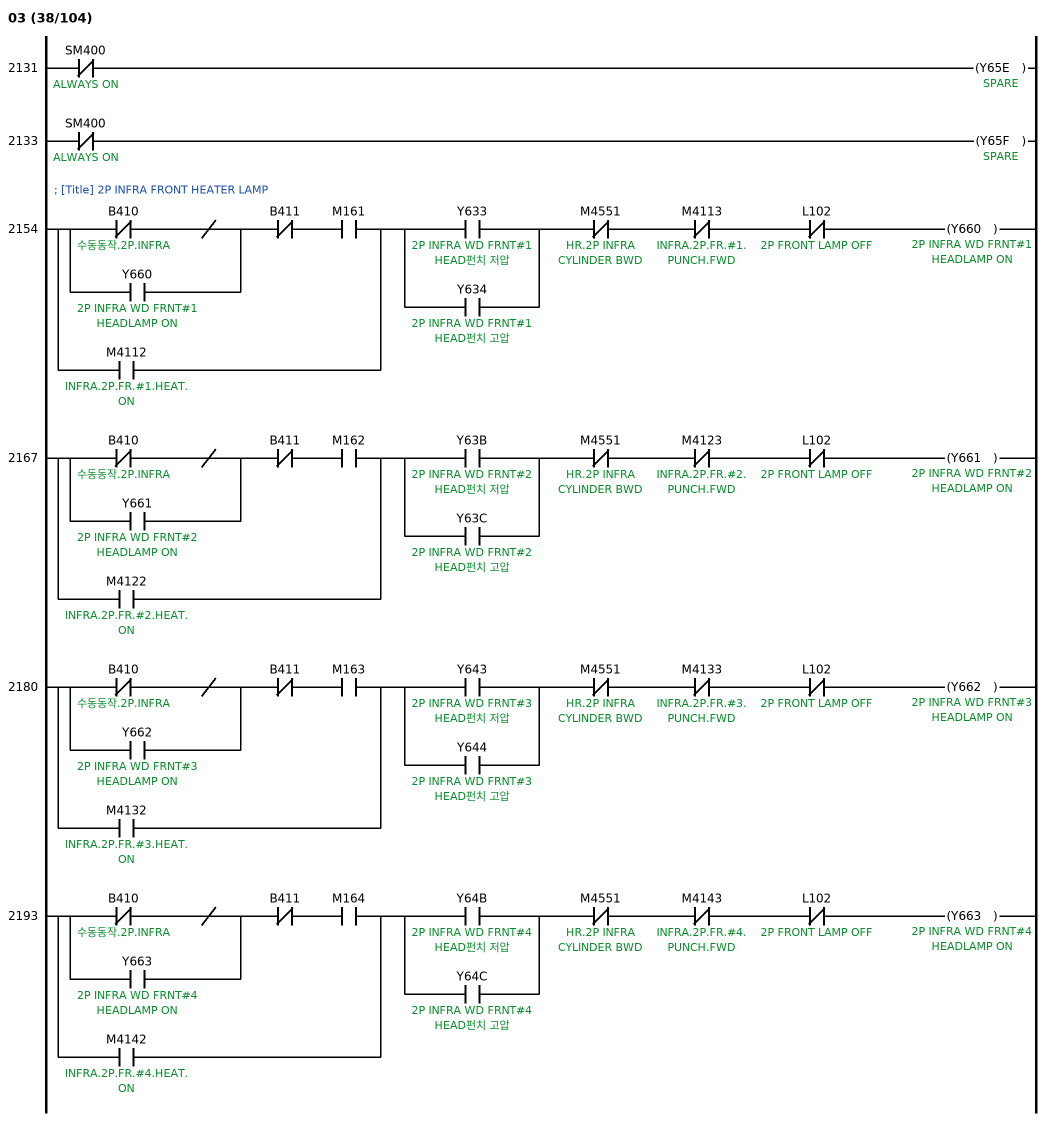
2131  LDI     SM400  ; ALWAYS ON
      OUT     Y65E  ; SPARE
2133  LDI     SM400  ; ALWAYS ON
      OUT     Y65F  ; SPARE
; [Title] 2P INFRA FRONT HEATER LAMP
2154  LDI     B410  ; 수동동작.2P.INFRA
      INV
      OR      Y660  ; 2P INFRA WD FRNT#1 HEADLAMP ON
      ANI     B411
      AND     M161
      OR      M4112  ; INFRA.2P.FR.#1.HEAT.ON
      LD      Y633  ; 2P INFRA WD FRNT#1 HEAD펀치 저압
      OR      Y634  ; 2P INFRA WD FRNT#1 HEAD펀치 고압
      ANB
      ANI     M4551  ; HR.2P INFRA CYLINDER BWD
      ANI     M4113  ; INFRA.2P.FR.#1.PUNCH.FWD
      ANI     L102  ; 2P FRONT LAMP OFF
      OUT     Y660  ; 2P INFRA WD FRNT#1 HEADLAMP ON
2167  LDI     B410  ; 수동동작.2P.INFRA
      INV
      OR      Y661  ; 2P INFRA WD FRNT#2 HEADLAMP ON
      ANI     B411
      AND     M162
      OR      M4122  ; INFRA.2P.FR.#2.HEAT.ON
      LD      Y63B  ; 2P INFRA WD FRNT#2 HEAD펀치 저압
      OR      Y63C  ; 2P INFRA WD FRNT#2 HEAD펀치 고압
      ANB
      ANI     M4551  ; HR.2P INFRA CYLINDER BWD
      ANI     M4123  ; INFRA.2P.FR.#2.PUNCH.FWD
      ANI     L102  ; 2P FRONT LAMP OFF
      OUT     Y661  ; 2P INFRA WD FRNT#2 HEADLAMP ON
2180  LDI     B410  ; 수동동작.2P.INFRA
      INV
      OR      Y662  ; 2P INFRA WD FRNT#3 HEADLAMP ON
      ANI     B411
      AND     M163
      OR      M4132  ; INFRA.2P.FR.#3.HEAT.ON
      LD      Y643  ; 2P INFRA WD FRNT#3 HEAD펀치 저압
      OR      Y644  ; 2P INFRA WD FRNT#3 HEAD펀치 고압
      ANB
      ANI     M4551  ; HR.2P INFRA CYLINDER BWD
      ANI     M4133  ; INFRA.2P.FR.#3.PUNCH.FWD
      ANI     L102  ; 2P FRONT LAMP OFF
      OUT     Y662  ; 2P INFRA WD FRNT#3 HEADLAMP ON
2193  LDI     B410  ; 수동동작.2P.INFRA
      INV
      OR      Y663  ; 2P INFRA WD FRNT#4 HEADLAMP ON
      ANI     B411
      AND     M164
      OR      M4142  ; INFRA.2P.FR.#4.HEAT.ON
      LD      Y64B  ; 2P INFRA WD FRNT#4 HEAD펀치 저압
      OR      Y64C  ; 2P INFRA WD FRNT#4 HEAD펀치 고압
      ANB
      ANI     M4551  ; HR.2P INFRA CYLINDER BWD
      ANI     M4143  ; INFRA.2P.FR.#4.PUNCH.FWD
      ANI     L102  ; 2P FRONT LAMP OFF
      OUT     Y663  ; 2P INFRA WD FRNT#4 HEADLAMP ON
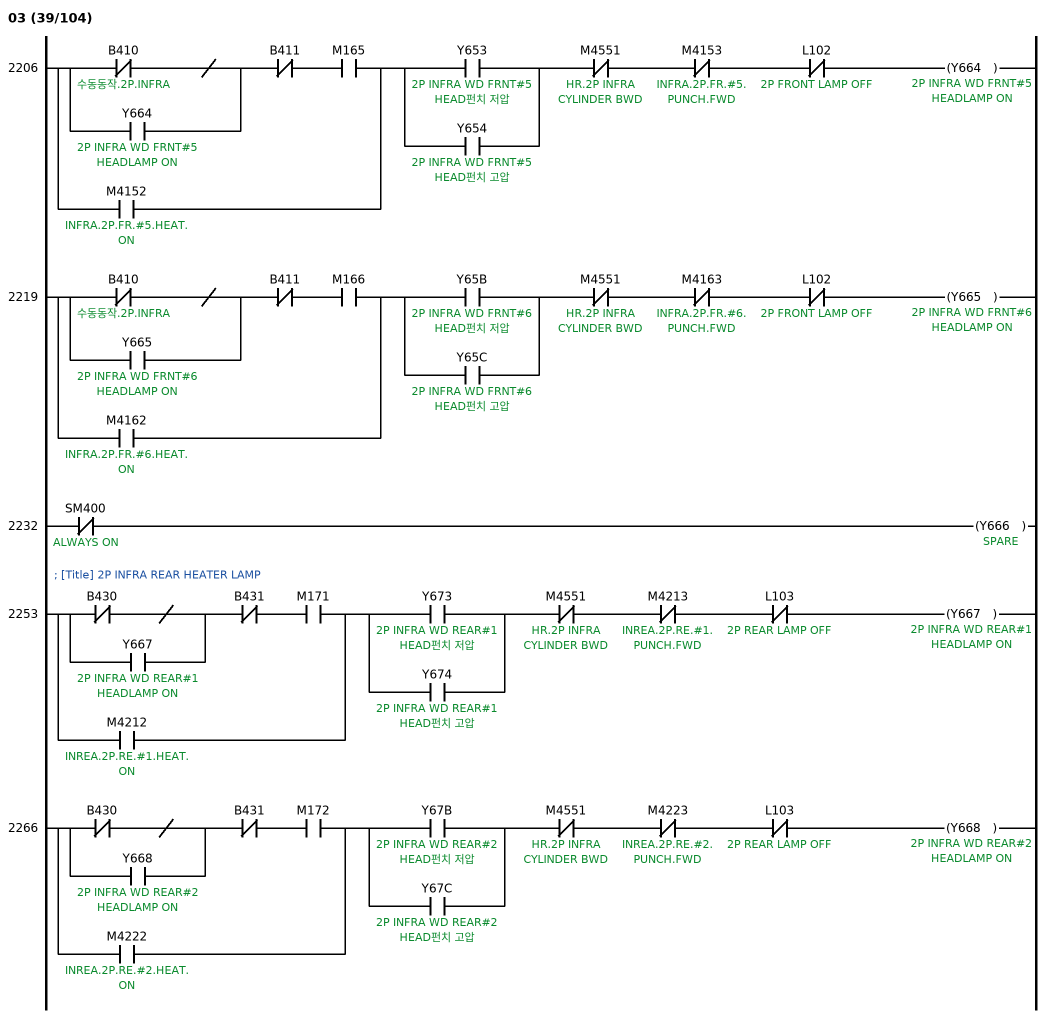
2206  LDI     B410  ; 수동동작.2P.INFRA
      INV
      OR      Y664  ; 2P INFRA WD FRNT#5 HEADLAMP ON
      ANI     B411
      AND     M165
      OR      M4152  ; INFRA.2P.FR.#5.HEAT.ON
      LD      Y653  ; 2P INFRA WD FRNT#5 HEAD펀치 저압
      OR      Y654  ; 2P INFRA WD FRNT#5 HEAD펀치 고압
      ANB
      ANI     M4551  ; HR.2P INFRA CYLINDER BWD
      ANI     M4153  ; INFRA.2P.FR.#5.PUNCH.FWD
      ANI     L102  ; 2P FRONT LAMP OFF
      OUT     Y664  ; 2P INFRA WD FRNT#5 HEADLAMP ON
2219  LDI     B410  ; 수동동작.2P.INFRA
      INV
      OR      Y665  ; 2P INFRA WD FRNT#6 HEADLAMP ON
      ANI     B411
      AND     M166
      OR      M4162  ; INFRA.2P.FR.#6.HEAT.ON
      LD      Y65B  ; 2P INFRA WD FRNT#6 HEAD펀치 저압
      OR      Y65C  ; 2P INFRA WD FRNT#6 HEAD펀치 고압
      ANB
      ANI     M4551  ; HR.2P INFRA CYLINDER BWD
      ANI     M4163  ; INFRA.2P.FR.#6.PUNCH.FWD
      ANI     L102  ; 2P FRONT LAMP OFF
      OUT     Y665  ; 2P INFRA WD FRNT#6 HEADLAMP ON
2232  LDI     SM400  ; ALWAYS ON
      OUT     Y666  ; SPARE
; [Title] 2P INFRA REAR HEATER LAMP
2253  LDI     B430
      INV
      OR      Y667  ; 2P INFRA WD REAR#1 HEADLAMP ON
      ANI     B431
      AND     M171
      OR      M4212  ; INREA.2P.RE.#1.HEAT.ON
      LD      Y673  ; 2P INFRA WD REAR#1 HEAD펀치 저압
      OR      Y674  ; 2P INFRA WD REAR#1 HEAD펀치 고압
      ANB
      ANI     M4551  ; HR.2P INFRA CYLINDER BWD
      ANI     M4213  ; INREA.2P.RE.#1.PUNCH.FWD
      ANI     L103  ; 2P REAR LAMP OFF
      OUT     Y667  ; 2P INFRA WD REAR#1 HEADLAMP ON
2266  LDI     B430
      INV
      OR      Y668  ; 2P INFRA WD REAR#2 HEADLAMP ON
      ANI     B431
      AND     M172
      OR      M4222  ; INREA.2P.RE.#2.HEAT.ON
      LD      Y67B  ; 2P INFRA WD REAR#2 HEAD펀치 저압
      OR      Y67C  ; 2P INFRA WD REAR#2 HEAD펀치 고압
      ANB
      ANI     M4551  ; HR.2P INFRA CYLINDER BWD
      ANI     M4223  ; INREA.2P.RE.#2.PUNCH.FWD
      ANI     L103  ; 2P REAR LAMP OFF
      OUT     Y668  ; 2P INFRA WD REAR#2 HEADLAMP ON
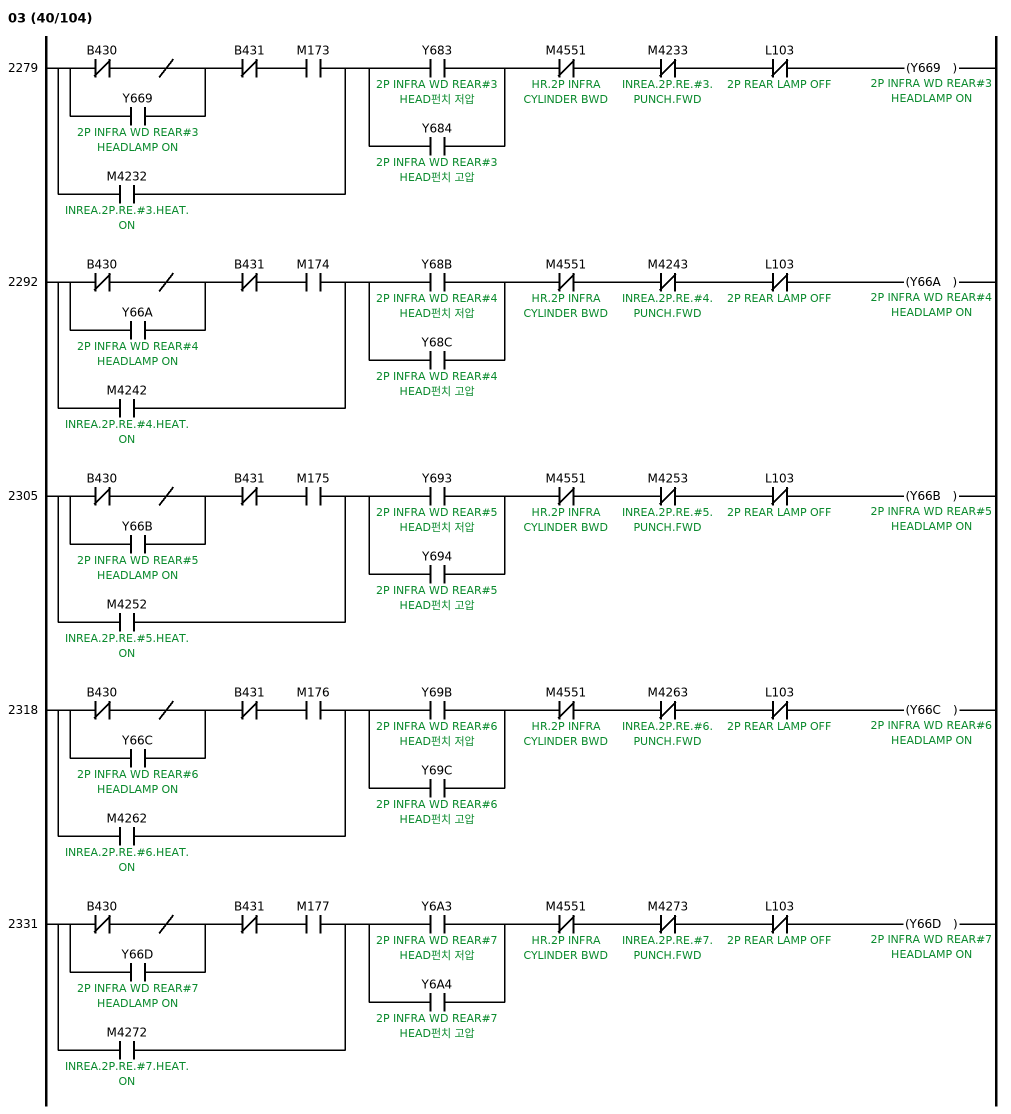
2279  LDI     B430
      INV
      OR      Y669  ; 2P INFRA WD REAR#3 HEADLAMP ON
      ANI     B431
      AND     M173
      OR      M4232  ; INREA.2P.RE.#3.HEAT.ON
      LD      Y683  ; 2P INFRA WD REAR#3 HEAD펀치 저압
      OR      Y684  ; 2P INFRA WD REAR#3 HEAD펀치 고압
      ANB
      ANI     M4551  ; HR.2P INFRA CYLINDER BWD
      ANI     M4233  ; INREA.2P.RE.#3.PUNCH.FWD
      ANI     L103  ; 2P REAR LAMP OFF
      OUT     Y669  ; 2P INFRA WD REAR#3 HEADLAMP ON
2292  LDI     B430
      INV
      OR      Y66A  ; 2P INFRA WD REAR#4 HEADLAMP ON
      ANI     B431
      AND     M174
      OR      M4242  ; INREA.2P.RE.#4.HEAT.ON
      LD      Y68B  ; 2P INFRA WD REAR#4 HEAD펀치 저압
      OR      Y68C  ; 2P INFRA WD REAR#4 HEAD펀치 고압
      ANB
      ANI     M4551  ; HR.2P INFRA CYLINDER BWD
      ANI     M4243  ; INREA.2P.RE.#4.PUNCH.FWD
      ANI     L103  ; 2P REAR LAMP OFF
      OUT     Y66A  ; 2P INFRA WD REAR#4 HEADLAMP ON
2305  LDI     B430
      INV
      OR      Y66B  ; 2P INFRA WD REAR#5 HEADLAMP ON
      ANI     B431
      AND     M175
      OR      M4252  ; INREA.2P.RE.#5.HEAT.ON
      LD      Y693  ; 2P INFRA WD REAR#5 HEAD펀치 저압
      OR      Y694  ; 2P INFRA WD REAR#5 HEAD펀치 고압
      ANB
      ANI     M4551  ; HR.2P INFRA CYLINDER BWD
      ANI     M4253  ; INREA.2P.RE.#5.PUNCH.FWD
      ANI     L103  ; 2P REAR LAMP OFF
      OUT     Y66B  ; 2P INFRA WD REAR#5 HEADLAMP ON
2318  LDI     B430
      INV
      OR      Y66C  ; 2P INFRA WD REAR#6 HEADLAMP ON
      ANI     B431
      AND     M176
      OR      M4262  ; INREA.2P.RE.#6.HEAT.ON
      LD      Y69B  ; 2P INFRA WD REAR#6 HEAD펀치 저압
      OR      Y69C  ; 2P INFRA WD REAR#6 HEAD펀치 고압
      ANB
      ANI     M4551  ; HR.2P INFRA CYLINDER BWD
      ANI     M4263  ; INREA.2P.RE.#6.PUNCH.FWD
      ANI     L103  ; 2P REAR LAMP OFF
      OUT     Y66C  ; 2P INFRA WD REAR#6 HEADLAMP ON
2331  LDI     B430
      INV
      OR      Y66D  ; 2P INFRA WD REAR#7 HEADLAMP ON
      ANI     B431
      AND     M177
      OR      M4272  ; INREA.2P.RE.#7.HEAT.ON
      LD      Y6A3  ; 2P INFRA WD REAR#7 HEAD펀치 저압
      OR      Y6A4  ; 2P INFRA WD REAR#7 HEAD펀치 고압
      ANB
      ANI     M4551  ; HR.2P INFRA CYLINDER BWD
      ANI     M4273  ; INREA.2P.RE.#7.PUNCH.FWD
      ANI     L103  ; 2P REAR LAMP OFF
      OUT     Y66D  ; 2P INFRA WD REAR#7 HEADLAMP ON
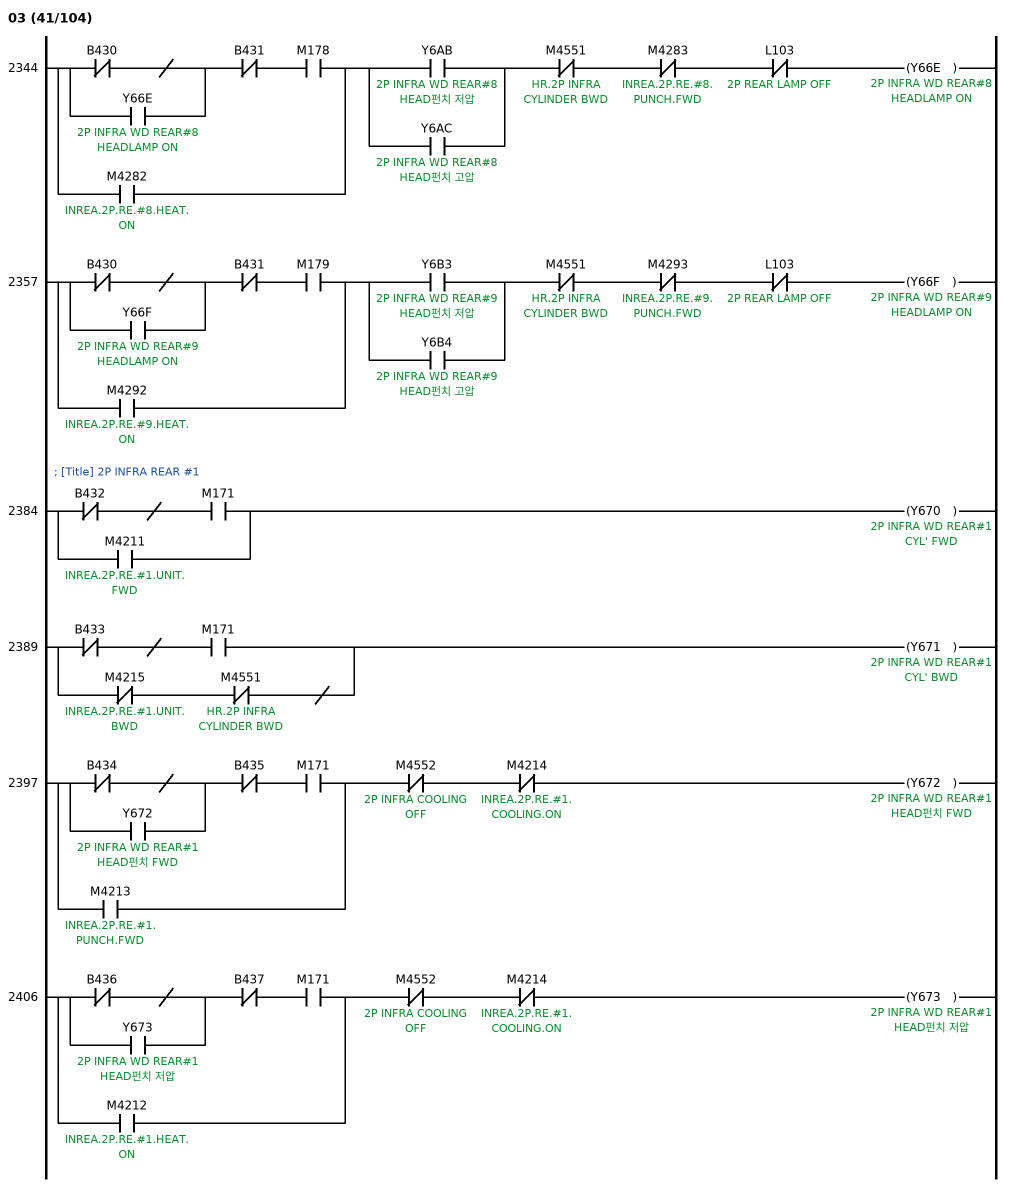
2344  LDI     B430
      INV
      OR      Y66E  ; 2P INFRA WD REAR#8 HEADLAMP ON
      ANI     B431
      AND     M178
      OR      M4282  ; INREA.2P.RE.#8.HEAT.ON
      LD      Y6AB  ; 2P INFRA WD REAR#8 HEAD펀치 저압
      OR      Y6AC  ; 2P INFRA WD REAR#8 HEAD펀치 고압
      ANB
      ANI     M4551  ; HR.2P INFRA CYLINDER BWD
      ANI     M4283  ; INREA.2P.RE.#8.PUNCH.FWD
      ANI     L103  ; 2P REAR LAMP OFF
      OUT     Y66E  ; 2P INFRA WD REAR#8 HEADLAMP ON
2357  LDI     B430
      INV
      OR      Y66F  ; 2P INFRA WD REAR#9 HEADLAMP ON
      ANI     B431
      AND     M179
      OR      M4292  ; INREA.2P.RE.#9.HEAT.ON
      LD      Y6B3  ; 2P INFRA WD REAR#9 HEAD펀치 저압
      OR      Y6B4  ; 2P INFRA WD REAR#9 HEAD펀치 고압
      ANB
      ANI     M4551  ; HR.2P INFRA CYLINDER BWD
      ANI     M4293  ; INREA.2P.RE.#9.PUNCH.FWD
      ANI     L103  ; 2P REAR LAMP OFF
      OUT     Y66F  ; 2P INFRA WD REAR#9 HEADLAMP ON
; [Title] 2P INFRA REAR #1
2384  LDI     B432
      INV
      AND     M171
      OR      M4211  ; INREA.2P.RE.#1.UNIT.FWD
      OUT     Y670  ; 2P INFRA WD REAR#1 CYL' FWD
2389  LDI     B433
      INV
      AND     M171
      LDI     M4215  ; INREA.2P.RE.#1.UNIT.BWD
      ANI     M4551  ; HR.2P INFRA CYLINDER BWD
      INV
      ORB
      OUT     Y671  ; 2P INFRA WD REAR#1 CYL' BWD
2397  LDI     B434
      INV
      OR      Y672  ; 2P INFRA WD REAR#1 HEAD펀치 FWD
      ANI     B435
      AND     M171
      OR      M4213  ; INREA.2P.RE.#1.PUNCH.FWD
      ANI     M4552  ; 2P INFRA COOLING OFF
      ANI     M4214  ; INREA.2P.RE.#1.COOLING.ON
      OUT     Y672  ; 2P INFRA WD REAR#1 HEAD펀치 FWD
2406  LDI     B436
      INV
      OR      Y673  ; 2P INFRA WD REAR#1 HEAD펀치 저압
      ANI     B437
      AND     M171
      OR      M4212  ; INREA.2P.RE.#1.HEAT.ON
      ANI     M4552  ; 2P INFRA COOLING OFF
      ANI     M4214  ; INREA.2P.RE.#1.COOLING.ON
      OUT     Y673  ; 2P INFRA WD REAR#1 HEAD펀치 저압
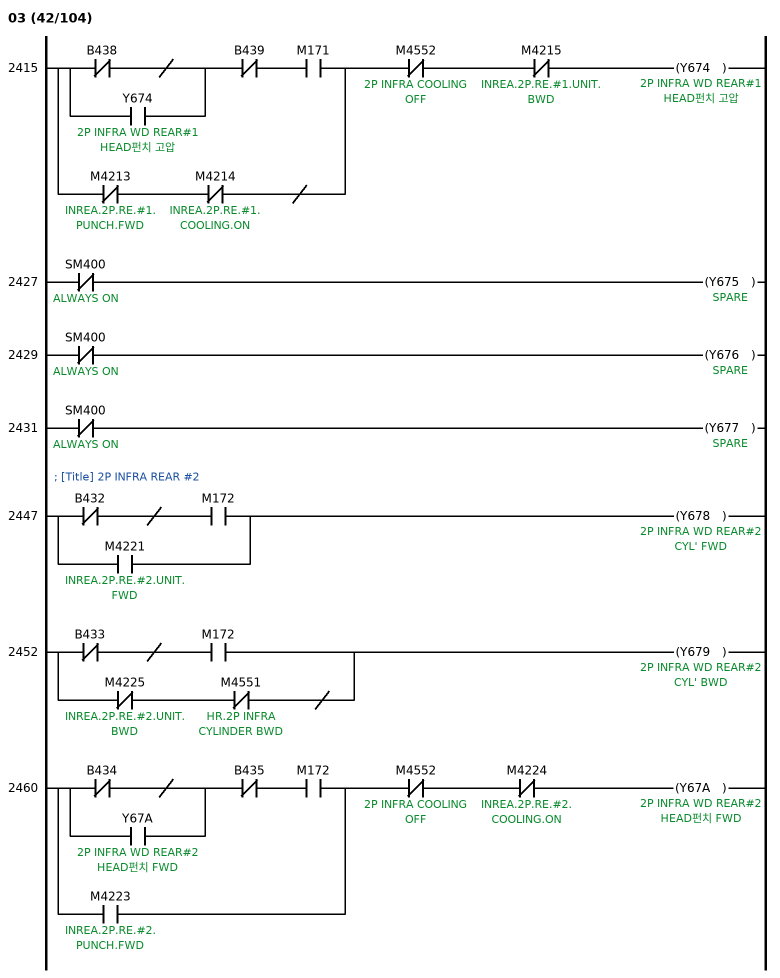
2415  LDI     B438
      INV
      OR      Y674  ; 2P INFRA WD REAR#1 HEAD펀치 고압
      ANI     B439
      AND     M171
      LDI     M4213  ; INREA.2P.RE.#1.PUNCH.FWD
      ANI     M4214  ; INREA.2P.RE.#1.COOLING.ON
      INV
      ORB
      ANI     M4552  ; 2P INFRA COOLING OFF
      ANI     M4215  ; INREA.2P.RE.#1.UNIT.BWD
      OUT     Y674  ; 2P INFRA WD REAR#1 HEAD펀치 고압
2427  LDI     SM400  ; ALWAYS ON
      OUT     Y675  ; SPARE
2429  LDI     SM400  ; ALWAYS ON
      OUT     Y676  ; SPARE
2431  LDI     SM400  ; ALWAYS ON
      OUT     Y677  ; SPARE
; [Title] 2P INFRA REAR #2
2447  LDI     B432
      INV
      AND     M172
      OR      M4221  ; INREA.2P.RE.#2.UNIT.FWD
      OUT     Y678  ; 2P INFRA WD REAR#2 CYL' FWD
2452  LDI     B433
      INV
      AND     M172
      LDI     M4225  ; INREA.2P.RE.#2.UNIT.BWD
      ANI     M4551  ; HR.2P INFRA CYLINDER BWD
      INV
      ORB
      OUT     Y679  ; 2P INFRA WD REAR#2 CYL' BWD
2460  LDI     B434
      INV
      OR      Y67A  ; 2P INFRA WD REAR#2 HEAD펀치 FWD
      ANI     B435
      AND     M172
      OR      M4223  ; INREA.2P.RE.#2.PUNCH.FWD
      ANI     M4552  ; 2P INFRA COOLING OFF
      ANI     M4224  ; INREA.2P.RE.#2.COOLING.ON
      OUT     Y67A  ; 2P INFRA WD REAR#2 HEAD펀치 FWD
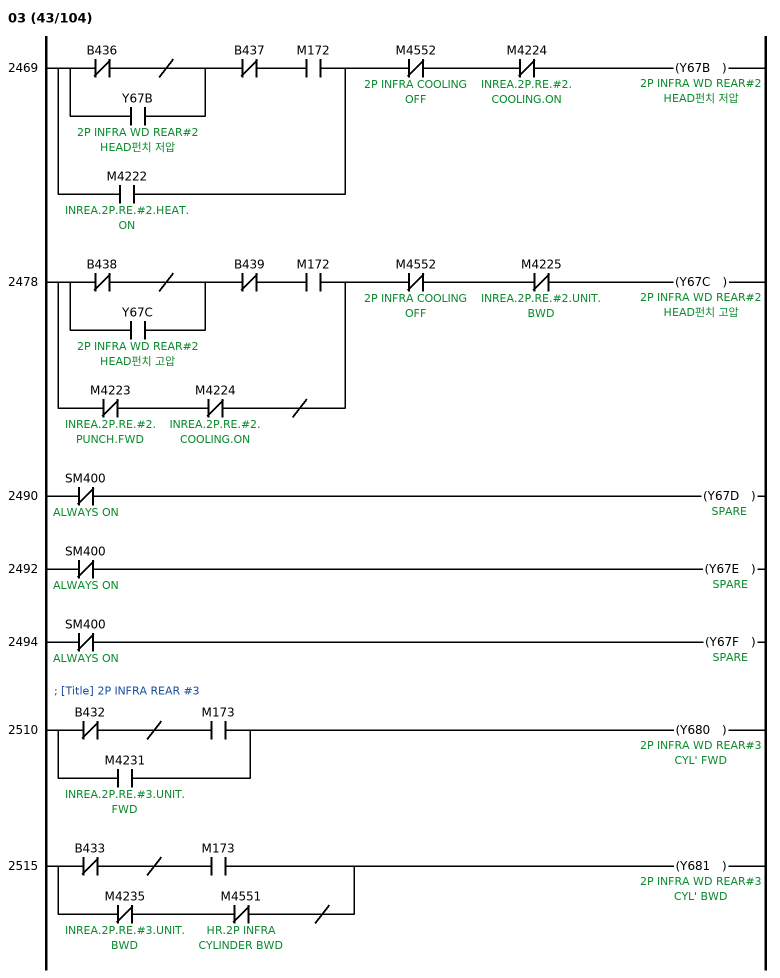
2469  LDI     B436
      INV
      OR      Y67B  ; 2P INFRA WD REAR#2 HEAD펀치 저압
      ANI     B437
      AND     M172
      OR      M4222  ; INREA.2P.RE.#2.HEAT.ON
      ANI     M4552  ; 2P INFRA COOLING OFF
      ANI     M4224  ; INREA.2P.RE.#2.COOLING.ON
      OUT     Y67B  ; 2P INFRA WD REAR#2 HEAD펀치 저압
2478  LDI     B438
      INV
      OR      Y67C  ; 2P INFRA WD REAR#2 HEAD펀치 고압
      ANI     B439
      AND     M172
      LDI     M4223  ; INREA.2P.RE.#2.PUNCH.FWD
      ANI     M4224  ; INREA.2P.RE.#2.COOLING.ON
      INV
      ORB
      ANI     M4552  ; 2P INFRA COOLING OFF
      ANI     M4225  ; INREA.2P.RE.#2.UNIT.BWD
      OUT     Y67C  ; 2P INFRA WD REAR#2 HEAD펀치 고압
2490  LDI     SM400  ; ALWAYS ON
      OUT     Y67D  ; SPARE
2492  LDI     SM400  ; ALWAYS ON
      OUT     Y67E  ; SPARE
2494  LDI     SM400  ; ALWAYS ON
      OUT     Y67F  ; SPARE
; [Title] 2P INFRA REAR #3
2510  LDI     B432
      INV
      AND     M173
      OR      M4231  ; INREA.2P.RE.#3.UNIT.FWD
      OUT     Y680  ; 2P INFRA WD REAR#3 CYL' FWD
2515  LDI     B433
      INV
      AND     M173
      LDI     M4235  ; INREA.2P.RE.#3.UNIT.BWD
      ANI     M4551  ; HR.2P INFRA CYLINDER BWD
      INV
      ORB
      OUT     Y681  ; 2P INFRA WD REAR#3 CYL' BWD
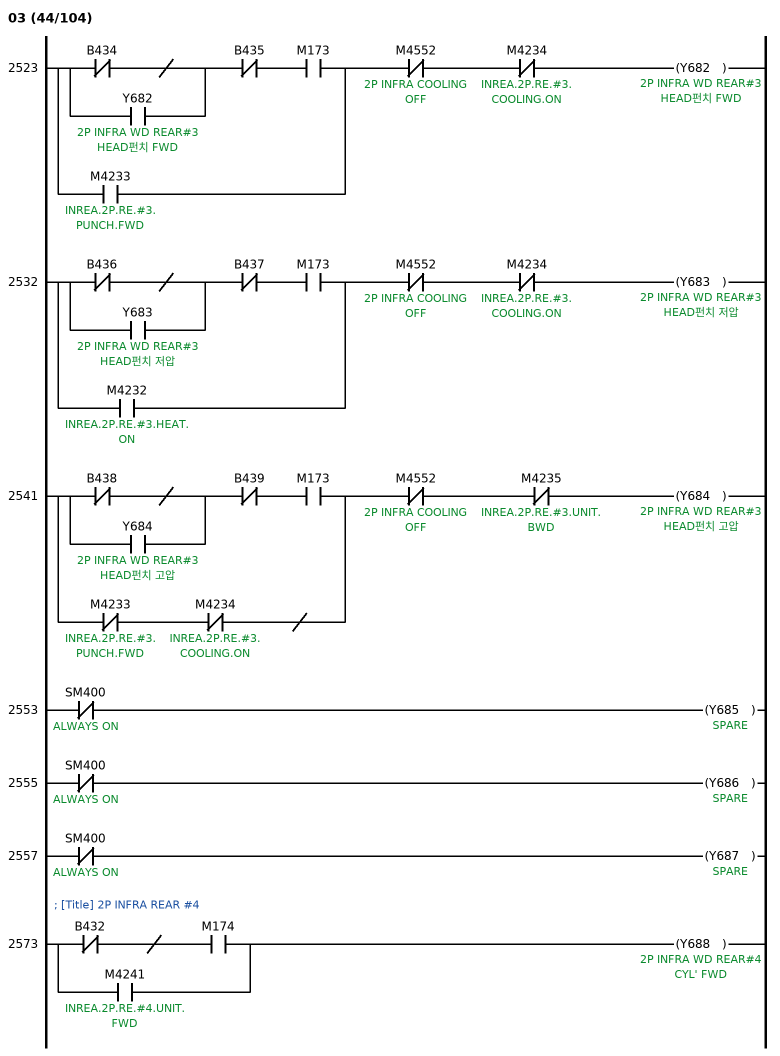
2523  LDI     B434
      INV
      OR      Y682  ; 2P INFRA WD REAR#3 HEAD펀치 FWD
      ANI     B435
      AND     M173
      OR      M4233  ; INREA.2P.RE.#3.PUNCH.FWD
      ANI     M4552  ; 2P INFRA COOLING OFF
      ANI     M4234  ; INREA.2P.RE.#3.COOLING.ON
      OUT     Y682  ; 2P INFRA WD REAR#3 HEAD펀치 FWD
2532  LDI     B436
      INV
      OR      Y683  ; 2P INFRA WD REAR#3 HEAD펀치 저압
      ANI     B437
      AND     M173
      OR      M4232  ; INREA.2P.RE.#3.HEAT.ON
      ANI     M4552  ; 2P INFRA COOLING OFF
      ANI     M4234  ; INREA.2P.RE.#3.COOLING.ON
      OUT     Y683  ; 2P INFRA WD REAR#3 HEAD펀치 저압
2541  LDI     B438
      INV
      OR      Y684  ; 2P INFRA WD REAR#3 HEAD펀치 고압
      ANI     B439
      AND     M173
      LDI     M4233  ; INREA.2P.RE.#3.PUNCH.FWD
      ANI     M4234  ; INREA.2P.RE.#3.COOLING.ON
      INV
      ORB
      ANI     M4552  ; 2P INFRA COOLING OFF
      ANI     M4235  ; INREA.2P.RE.#3.UNIT.BWD
      OUT     Y684  ; 2P INFRA WD REAR#3 HEAD펀치 고압
2553  LDI     SM400  ; ALWAYS ON
      OUT     Y685  ; SPARE
2555  LDI     SM400  ; ALWAYS ON
      OUT     Y686  ; SPARE
2557  LDI     SM400  ; ALWAYS ON
      OUT     Y687  ; SPARE
; [Title] 2P INFRA REAR #4
2573  LDI     B432
      INV
      AND     M174
      OR      M4241  ; INREA.2P.RE.#4.UNIT.FWD
      OUT     Y688  ; 2P INFRA WD REAR#4 CYL' FWD
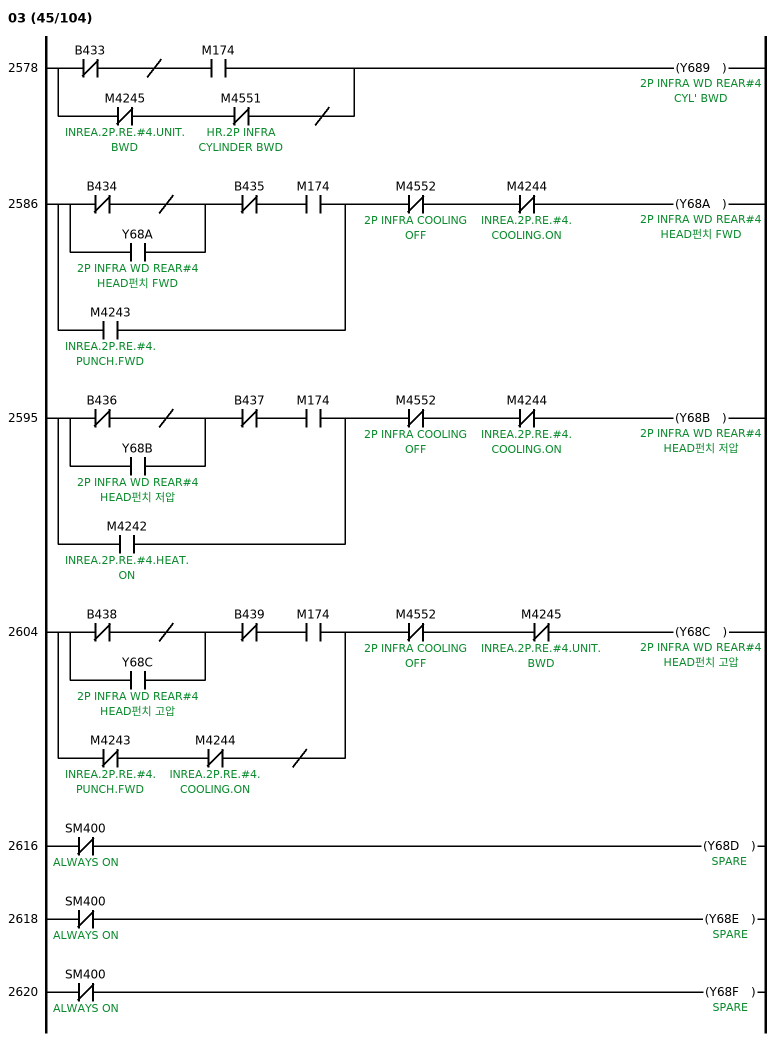
2578  LDI     B433
      INV
      AND     M174
      LDI     M4245  ; INREA.2P.RE.#4.UNIT.BWD
      ANI     M4551  ; HR.2P INFRA CYLINDER BWD
      INV
      ORB
      OUT     Y689  ; 2P INFRA WD REAR#4 CYL' BWD
2586  LDI     B434
      INV
      OR      Y68A  ; 2P INFRA WD REAR#4 HEAD펀치 FWD
      ANI     B435
      AND     M174
      OR      M4243  ; INREA.2P.RE.#4.PUNCH.FWD
      ANI     M4552  ; 2P INFRA COOLING OFF
      ANI     M4244  ; INREA.2P.RE.#4.COOLING.ON
      OUT     Y68A  ; 2P INFRA WD REAR#4 HEAD펀치 FWD
2595  LDI     B436
      INV
      OR      Y68B  ; 2P INFRA WD REAR#4 HEAD펀치 저압
      ANI     B437
      AND     M174
      OR      M4242  ; INREA.2P.RE.#4.HEAT.ON
      ANI     M4552  ; 2P INFRA COOLING OFF
      ANI     M4244  ; INREA.2P.RE.#4.COOLING.ON
      OUT     Y68B  ; 2P INFRA WD REAR#4 HEAD펀치 저압
2604  LDI     B438
      INV
      OR      Y68C  ; 2P INFRA WD REAR#4 HEAD펀치 고압
      ANI     B439
      AND     M174
      LDI     M4243  ; INREA.2P.RE.#4.PUNCH.FWD
      ANI     M4244  ; INREA.2P.RE.#4.COOLING.ON
      INV
      ORB
      ANI     M4552  ; 2P INFRA COOLING OFF
      ANI     M4245  ; INREA.2P.RE.#4.UNIT.BWD
      OUT     Y68C  ; 2P INFRA WD REAR#4 HEAD펀치 고압
2616  LDI     SM400  ; ALWAYS ON
      OUT     Y68D  ; SPARE
2618  LDI     SM400  ; ALWAYS ON
      OUT     Y68E  ; SPARE
2620  LDI     SM400  ; ALWAYS ON
      OUT     Y68F  ; SPARE
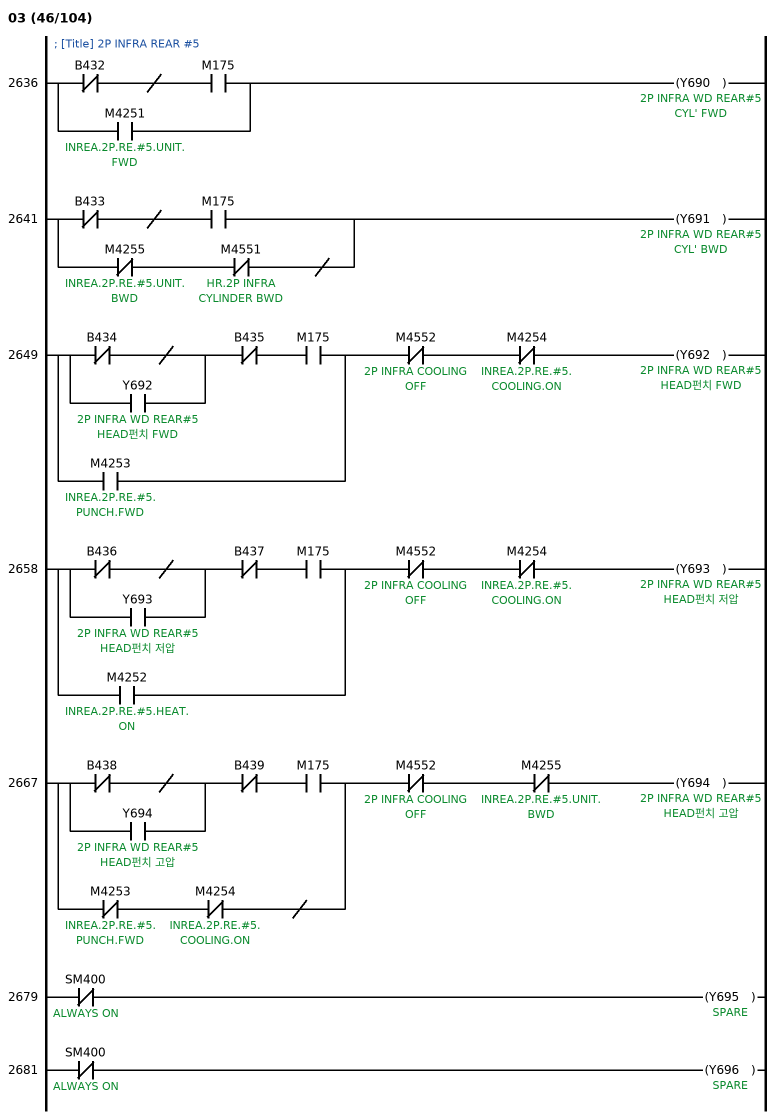
; [Title] 2P INFRA REAR #5
2636  LDI     B432
      INV
      AND     M175
      OR      M4251  ; INREA.2P.RE.#5.UNIT.FWD
      OUT     Y690  ; 2P INFRA WD REAR#5 CYL' FWD
2641  LDI     B433
      INV
      AND     M175
      LDI     M4255  ; INREA.2P.RE.#5.UNIT.BWD
      ANI     M4551  ; HR.2P INFRA CYLINDER BWD
      INV
      ORB
      OUT     Y691  ; 2P INFRA WD REAR#5 CYL' BWD
2649  LDI     B434
      INV
      OR      Y692  ; 2P INFRA WD REAR#5 HEAD펀치 FWD
      ANI     B435
      AND     M175
      OR      M4253  ; INREA.2P.RE.#5.PUNCH.FWD
      ANI     M4552  ; 2P INFRA COOLING OFF
      ANI     M4254  ; INREA.2P.RE.#5.COOLING.ON
      OUT     Y692  ; 2P INFRA WD REAR#5 HEAD펀치 FWD
2658  LDI     B436
      INV
      OR      Y693  ; 2P INFRA WD REAR#5 HEAD펀치 저압
      ANI     B437
      AND     M175
      OR      M4252  ; INREA.2P.RE.#5.HEAT.ON
      ANI     M4552  ; 2P INFRA COOLING OFF
      ANI     M4254  ; INREA.2P.RE.#5.COOLING.ON
      OUT     Y693  ; 2P INFRA WD REAR#5 HEAD펀치 저압
2667  LDI     B438
      INV
      OR      Y694  ; 2P INFRA WD REAR#5 HEAD펀치 고압
      ANI     B439
      AND     M175
      LDI     M4253  ; INREA.2P.RE.#5.PUNCH.FWD
      ANI     M4254  ; INREA.2P.RE.#5.COOLING.ON
      INV
      ORB
      ANI     M4552  ; 2P INFRA COOLING OFF
      ANI     M4255  ; INREA.2P.RE.#5.UNIT.BWD
      OUT     Y694  ; 2P INFRA WD REAR#5 HEAD펀치 고압
2679  LDI     SM400  ; ALWAYS ON
      OUT     Y695  ; SPARE
2681  LDI     SM400  ; ALWAYS ON
      OUT     Y696  ; SPARE
